(* IEC 61131-3 sources: verifaps-lib/geteta/examples/RTT_if, 5 files *)

(* ---- Preamble.st ---- *)
TYPE
    Magazin_states_t : (Green_Lamp , Init , Interstep , Magazin_Init , Magazin_Init_2 , Slider_Move_Back , Start_Magazin , Step0 , Step1 , convey);
    Stamp_states_t : (Green_Lamp , Init , Interstep , Interstep_2 , StampProcess , StampSliderBack , StampSliderForward , Stamp_Init_1 , Stamp_Init_2 , Stamp_Init_3 , Stamp_Init_4 , Start_Stamp , Step0 , Step1 , Step2);
    Crane_states_t : (Crane_Go_Up , Crane_Init , Crane_Init_2 , Crane_Lift_At_Stamp , Crane_Lift_Conveyor , Crane_Lift_Conveyor_Black , Crane_Lift_Magazin , Crane_Lift_Magazin_Metallic , Crane_Lift_NOT_Metallic_Black , Crane_Lower , Crane_On_Conveyor , Crane_On_Conveyor_Metallic , Crane_On_Conveyor_Not_Metallica_Black , Crane_On_Stamp_Metallic , Crane_On_Stamp_Stop_Black , Crane_Turn_Left_Back_To_Stamp , Crane_Turn_Left_From_Stamp , Crane_Turn_Left_Metallic , Crane_Turn_Left_NOT_Metallic , Crane_Turn_Left_NOT_Metallic_Black , Init , Interstep , Interstep_2 , Last_Workpiece_At_Stamp , Lower_Crane , Magazin_Stop , Magazin_Stop_Black , No_Workpiece_ready , Reset_interconnect , Start_Crane , Step0 , Suck_At_Stamp , TimeDelay , Turn_Right , Turn_Right_Black , pause , release , release_Black , release_Workpiece);
END_TYPE

(* ---- Code_13.st ---- *)
FUNCTION_BLOCK Main

VAR_OUTPUT  Actuator_AnalogCranePressure : INT; END_VAR
VAR_OUTPUT  Actuator_CraneLower : BOOL; END_VAR
VAR_OUTPUT  Actuator_CraneTurnClockwise : BOOL; END_VAR
VAR_OUTPUT  Actuator_CraneTurnCounterclockwise : BOOL; END_VAR
VAR_OUTPUT  Actuator_MagazinGreenLamp : BOOL; END_VAR
VAR_OUTPUT  Actuator_MagazinSlider : BOOL; END_VAR
VAR_OUTPUT  Actuator_MagazinVacuumOff : BOOL; END_VAR
VAR_OUTPUT  Actuator_MagazinVacuumOn : BOOL; END_VAR
VAR_OUTPUT  Actuator_MagazinWhiteLamp : BOOL; END_VAR
VAR_OUTPUT  Actuator_PusherY1 : BOOL; END_VAR
VAR_OUTPUT  Actuator_PusherY2 : BOOL; END_VAR
VAR_OUTPUT  Actuator_SorterConveyorTowardsCrane : BOOL; END_VAR
VAR_OUTPUT  Actuator_SorterConveyorTowardsStacker : BOOL; END_VAR
VAR_OUTPUT  Actuator_SorterGreenLampConveyor : BOOL; END_VAR
VAR_OUTPUT  Actuator_SorterWhiteLampConveyor : BOOL; END_VAR
VAR_OUTPUT  Actuator_StampGreenLamp : BOOL; END_VAR
VAR_OUTPUT  Actuator_StampPusher : BOOL; END_VAR
VAR_OUTPUT  Actuator_StampSliderMovedIn : BOOL; END_VAR
VAR_OUTPUT  Actuator_StampSliderMovedOut : BOOL; END_VAR
VAR_OUTPUT  Actuator_StampWhiteLamp : BOOL; END_VAR
VAR  Conveyor$Duration_Conveyor_Runtime : UINT := UINT#1125; END_VAR
VAR  Conveyor$Duration_Conveyor_Test : UINT := UINT#250; END_VAR
VAR  Conveyor$SFCInit : BOOL; END_VAR
VAR  Conveyor$SFCReset : BOOL; END_VAR
VAR  Conveyor$SorterConveyorTowardsCrane : BOOL; END_VAR
VAR  Conveyor$SorterConveyorTowardsStacker : BOOL; END_VAR
VAR  Conveyor$SorterGreenLampConveyor : BOOL; END_VAR
VAR  Conveyor$SorterLightbarrierCraneInterface : BOOL; END_VAR
VAR  Conveyor$SorterStartButton : BOOL; END_VAR
VAR  Conveyor$SorterSwitchManuellAutomatic : BOOL; END_VAR
VAR  Conveyor$SorterWhiteLampConveyor : BOOL; END_VAR
VAR  Conveyor$StartCommandConveyor : BOOL; END_VAR
VAR  Conveyor$StartVar : BOOL; END_VAR
VAR  Conveyor$Timer_Conveyor_Runtime$ET : USINT; END_VAR
VAR  Conveyor$Timer_Conveyor_Runtime$IN : BOOL; END_VAR
VAR  Conveyor$Timer_Conveyor_Runtime$PT : USINT; END_VAR
VAR  Conveyor$Timer_Conveyor_Runtime$Q : BOOL; END_VAR
VAR  Conveyor$Timer_Conveyor_Test$ET : USINT; END_VAR
VAR  Conveyor$Timer_Conveyor_Test$IN : BOOL; END_VAR
VAR  Conveyor$Timer_Conveyor_Test$PT : USINT; END_VAR
VAR  Conveyor$Timer_Conveyor_Test$Q : BOOL; END_VAR
VAR  Conveyor$_state : Conveyor_states_t; END_VAR
VAR  Conveyor$_transit : BOOL; END_VAR
VAR  Conveyor$interconnectConveyorStartCommand : BOOL; END_VAR
VAR  Conveyor$interconnectConveyorTerminationCommand : BOOL; END_VAR
VAR  Conveyor$interconnect_Conveyor_Runtime : BOOL; END_VAR
VAR  Conveyor$interconnect_Conveyor_Test : BOOL; END_VAR
VAR  Crane$AnalogCranePosition : INT; END_VAR
VAR  Crane$AnalogCranePressure : INT; END_VAR
VAR  Crane$CraneDown : BOOL; END_VAR
VAR  Crane$CraneLower : BOOL; END_VAR
VAR  Crane$CraneSucked : BOOL; END_VAR
VAR  Crane$CraneTurnClockwise : BOOL; END_VAR
VAR  Crane$CraneTurnCounterclockwise : BOOL; END_VAR
VAR  Crane$CraneUp : BOOL; END_VAR
VAR  Crane$Duration1 : UINT := UINT#375; END_VAR
VAR  Crane$MagazinCapacitiveSensor : BOOL; END_VAR
VAR  Crane$MagazinOpticalSensor : BOOL; END_VAR
VAR  Crane$MagazinSlider : BOOL; END_VAR
VAR  Crane$MagazinVacuumOff : BOOL; END_VAR
VAR  Crane$MagazinVacuumOn : BOOL; END_VAR
VAR  Crane$SFCInit : BOOL; END_VAR
VAR  Crane$SFCReset : BOOL; END_VAR
VAR  Crane$SliderMovedOut : BOOL; END_VAR
VAR  Crane$SliderNotMovedOut : BOOL; END_VAR
VAR  Crane$StampLowered : BOOL; END_VAR
VAR  Crane$StampSliderFilled : BOOL; END_VAR
VAR  Crane$StampSliderSensorMovedOut : BOOL; END_VAR
VAR  Crane$StartButtonMagazin : BOOL; END_VAR
VAR  Crane$StartCommandCrane : BOOL; END_VAR
VAR  Crane$StartVar : BOOL; END_VAR
VAR  Crane$TimeDelay_Timer$ET : USINT; END_VAR
VAR  Crane$TimeDelay_Timer$IN : BOOL; END_VAR
VAR  Crane$TimeDelay_Timer$PT : USINT; END_VAR
VAR  Crane$TimeDelay_Timer$Q : BOOL; END_VAR
VAR  Crane$TimeDelay_Timer_Duration : UINT := UINT#12; END_VAR
VAR  Crane$TimeDelay_Timer_interconnect : BOOL; END_VAR
VAR  Crane$Timer1$ET : USINT; END_VAR
VAR  Crane$Timer1$IN : BOOL; END_VAR
VAR  Crane$Timer1$PT : USINT; END_VAR
VAR  Crane$Timer1$Q : BOOL; END_VAR
VAR  Crane$WorkpieceReady : BOOL; END_VAR
VAR  Crane$_state : Crane_states_t; END_VAR
VAR  Crane$_transit : BOOL; END_VAR
VAR  Crane$actualtime1 : INT; END_VAR
VAR  Crane$interconnect : BOOL; END_VAR
VAR  Crane$interconnectCraneStartCommand : BOOL; END_VAR
VAR  Mag$AnalogCranePosition : INT; END_VAR
VAR  Mag$CraneDown : BOOL; END_VAR
VAR  Mag$CraneLower : BOOL; END_VAR
VAR  Mag$CraneOnConveyor : BOOL; END_VAR
VAR  Mag$CraneOnMagazin : BOOL; END_VAR
VAR  Mag$CraneSucked : BOOL; END_VAR
VAR  Mag$CraneTurnClockwise : BOOL; END_VAR
VAR  Mag$CraneTurnCounterclockwise : BOOL; END_VAR
VAR  Mag$CraneUp : BOOL; END_VAR
VAR  Mag$MagazinGreenLamp : BOOL; END_VAR
VAR  Mag$MagazinSlider : BOOL; END_VAR
VAR  Mag$MagazinVacuumOff : BOOL; END_VAR
VAR  Mag$MagazinVacuumOn : BOOL; END_VAR
VAR  Mag$MagazinWhiteLamp : BOOL; END_VAR
VAR  Mag$SFCInit : BOOL; END_VAR
VAR  Mag$SFCReset : BOOL; END_VAR
VAR  Mag$SliderMovedOut : BOOL; END_VAR
VAR  Mag$SliderNotMovedOut : BOOL; END_VAR
VAR  Mag$StartButtonMagazin : BOOL; END_VAR
VAR  Mag$StartCommandMagazin : BOOL; END_VAR
VAR  Mag$StartVar : BOOL; END_VAR
VAR  Mag$WorkpieceReady : BOOL; END_VAR
VAR  Mag$_state : Magazin_states_t; END_VAR
VAR  Mag$_transit : BOOL; END_VAR
VAR  Mag$interconnectMagazinStartCommand : BOOL; END_VAR
VAR  Pusher$Duration2 : UINT := UINT#500; END_VAR
VAR  Pusher$Duration3 : UINT := UINT#50; END_VAR
VAR  Pusher$Duration_Slide1_Black : UINT := UINT#237; END_VAR
VAR  Pusher$Duration_Slide1_Metal : UINT := UINT#75; END_VAR
VAR  Pusher$Duration_Slide1_White : UINT := UINT#75; END_VAR
VAR  Pusher$Duration_Slide2_Black : UINT := UINT#500; END_VAR
VAR  Pusher$Duration_Slide2_Metal : UINT := UINT#92; END_VAR
VAR  Pusher$Duration_Slide2_White : UINT := UINT#92; END_VAR
VAR  Pusher$Priority_Var_Black : INT := INT#3; END_VAR
VAR  Pusher$Priority_Var_Metal : INT := INT#3; END_VAR
VAR  Pusher$Priority_Var_White : INT := INT#3; END_VAR
VAR  Pusher$PusherY1 : BOOL; END_VAR
VAR  Pusher$PusherY2 : BOOL; END_VAR
VAR  Pusher$SFCInit : BOOL; END_VAR
VAR  Pusher$SFCReset : BOOL; END_VAR
VAR  Pusher$Slide1_black : INT := INT#1; END_VAR
VAR  Pusher$Slide1_metal : INT := INT#1; END_VAR
VAR  Pusher$Slide1_white : INT := INT#1; END_VAR
VAR  Pusher$Slide2_black : INT := INT#1; END_VAR
VAR  Pusher$Slide2_metal : INT := INT#1; END_VAR
VAR  Pusher$Slide2_white : INT := INT#1; END_VAR
VAR  Pusher$Slide3_black : INT := INT#1; END_VAR
VAR  Pusher$Slide3_metal : INT := INT#1; END_VAR
VAR  Pusher$Slide3_white : INT := INT#1; END_VAR
VAR  Pusher$SorterCapacitiveSensorPusher1 : BOOL; END_VAR
VAR  Pusher$SorterCapacitiveSensorPusher2 : BOOL; END_VAR
VAR  Pusher$SorterLightbarrierCraneInterface : BOOL; END_VAR
VAR  Pusher$SorterLightnessSensorPusher1 : BOOL; END_VAR
VAR  Pusher$SorterLightnessSensorPusher2 : BOOL; END_VAR
VAR  Pusher$SorterLightnessSensorPusher3 : BOOL; END_VAR
VAR  Pusher$SorterLightnesssensorCraneInterfaceInverse : BOOL; END_VAR
VAR  Pusher$SorterPusher1MovedIn : BOOL; END_VAR
VAR  Pusher$SorterPusher1MovedOut : BOOL; END_VAR
VAR  Pusher$SorterPusher2MovedIn : BOOL; END_VAR
VAR  Pusher$SorterPusher2MovedOut : BOOL; END_VAR
VAR  Pusher$SorterStartButton : BOOL; END_VAR
VAR  Pusher$StartVar : BOOL; END_VAR
VAR  Pusher$Timer2$ET : USINT; END_VAR
VAR  Pusher$Timer2$IN : BOOL; END_VAR
VAR  Pusher$Timer2$PT : USINT; END_VAR
VAR  Pusher$Timer2$Q : BOOL; END_VAR
VAR  Pusher$Timer3$ET : USINT; END_VAR
VAR  Pusher$Timer3$IN : BOOL; END_VAR
VAR  Pusher$Timer3$PT : USINT; END_VAR
VAR  Pusher$Timer3$Q : BOOL; END_VAR
VAR  Pusher$Timer_Slide1_Black$ET : USINT; END_VAR
VAR  Pusher$Timer_Slide1_Black$IN : BOOL; END_VAR
VAR  Pusher$Timer_Slide1_Black$PT : USINT; END_VAR
VAR  Pusher$Timer_Slide1_Black$Q : BOOL; END_VAR
VAR  Pusher$Timer_Slide1_Metal$ET : USINT; END_VAR
VAR  Pusher$Timer_Slide1_Metal$IN : BOOL; END_VAR
VAR  Pusher$Timer_Slide1_Metal$PT : USINT; END_VAR
VAR  Pusher$Timer_Slide1_Metal$Q : BOOL; END_VAR
VAR  Pusher$Timer_Slide1_White$ET : USINT; END_VAR
VAR  Pusher$Timer_Slide1_White$IN : BOOL; END_VAR
VAR  Pusher$Timer_Slide1_White$PT : USINT; END_VAR
VAR  Pusher$Timer_Slide1_White$Q : BOOL; END_VAR
VAR  Pusher$Timer_Slide2_Black$ET : USINT; END_VAR
VAR  Pusher$Timer_Slide2_Black$IN : BOOL; END_VAR
VAR  Pusher$Timer_Slide2_Black$PT : USINT; END_VAR
VAR  Pusher$Timer_Slide2_Black$Q : BOOL; END_VAR
VAR  Pusher$Timer_Slide2_Metal$ET : USINT; END_VAR
VAR  Pusher$Timer_Slide2_Metal$IN : BOOL; END_VAR
VAR  Pusher$Timer_Slide2_Metal$PT : USINT; END_VAR
VAR  Pusher$Timer_Slide2_Metal$Q : BOOL; END_VAR
VAR  Pusher$Timer_Slide2_White$ET : USINT; END_VAR
VAR  Pusher$Timer_Slide2_White$IN : BOOL; END_VAR
VAR  Pusher$Timer_Slide2_White$PT : USINT; END_VAR
VAR  Pusher$Timer_Slide2_White$Q : BOOL; END_VAR
VAR  Pusher$_state : Pusher_states_t; END_VAR
VAR  Pusher$_transit : BOOL; END_VAR
VAR  Pusher$interconnect2 : BOOL; END_VAR
VAR  Pusher$interconnect3 : BOOL; END_VAR
VAR  Pusher$interconnect_Slide1_Black : BOOL; END_VAR
VAR  Pusher$interconnect_Slide1_Metal : BOOL; END_VAR
VAR  Pusher$interconnect_Slide1_White : BOOL; END_VAR
VAR  Pusher$interconnect_Slide2_Black : BOOL; END_VAR
VAR  Pusher$interconnect_Slide2_Metal : BOOL; END_VAR
VAR  Pusher$interconnect_Slide2_White : BOOL; END_VAR
VAR_INPUT  Sensor_AnalogCranePosition : INT; END_VAR
VAR_INPUT  Sensor_CraneDown : BOOL; END_VAR
VAR_INPUT  Sensor_CraneOnConveyor : BOOL; END_VAR
VAR_INPUT  Sensor_CraneOnMagazin : BOOL; END_VAR
VAR_INPUT  Sensor_CranePosition : BOOL; END_VAR
VAR_INPUT  Sensor_CranePositionStamp : BOOL; END_VAR
VAR_INPUT  Sensor_CraneSucked : BOOL; END_VAR
VAR_INPUT  Sensor_CraneUp : BOOL; END_VAR
VAR_INPUT  Sensor_MagazinCapacitiveSensor : BOOL; END_VAR
VAR_INPUT  Sensor_MagazinEmergencyStop : BOOL; END_VAR
VAR_INPUT  Sensor_MagazinOpticalSensor : BOOL; END_VAR
VAR_INPUT  Sensor_MagazinSwitchManuellAutomatic : BOOL; END_VAR
VAR_INPUT  Sensor_SliderMovedOut : BOOL; END_VAR
VAR_INPUT  Sensor_SliderNotMovedOut : BOOL; END_VAR
VAR_INPUT  Sensor_SorterCapacitiveSensorPusher1 : BOOL; END_VAR
VAR_INPUT  Sensor_SorterCapacitiveSensorPusher2 : BOOL; END_VAR
VAR_INPUT  Sensor_SorterEmergencyStop : BOOL; END_VAR
VAR_INPUT  Sensor_SorterLightbarrierCraneInterface : BOOL; END_VAR
VAR_INPUT  Sensor_SorterLightnessSensorPusher1 : BOOL; END_VAR
VAR_INPUT  Sensor_SorterLightnessSensorPusher2 : BOOL; END_VAR
VAR_INPUT  Sensor_SorterLightnessSensorPusher3 : BOOL; END_VAR
VAR_INPUT  Sensor_SorterLightnesssensorCraneInterfaceInverse : BOOL; END_VAR
VAR_INPUT  Sensor_SorterPusher1MovedIn : BOOL; END_VAR
VAR_INPUT  Sensor_SorterPusher1MovedOut : BOOL; END_VAR
VAR_INPUT  Sensor_SorterPusher2MovedIn : BOOL; END_VAR
VAR_INPUT  Sensor_SorterPusher2MovedOut : BOOL; END_VAR
VAR_INPUT  Sensor_SorterStartButton : BOOL; END_VAR
VAR_INPUT  Sensor_SorterSwitchManuellAutomatic : BOOL; END_VAR
VAR_INPUT  Sensor_StampEmergencyStop : BOOL; END_VAR
VAR_INPUT  Sensor_StampLowered : BOOL; END_VAR
VAR_INPUT  Sensor_StampSliderFilled : BOOL; END_VAR
VAR_INPUT  Sensor_StampSliderSensorMovedIn : BOOL; END_VAR
VAR_INPUT  Sensor_StampSliderSensorMovedOut : BOOL; END_VAR
VAR_INPUT  Sensor_StampStartButton : BOOL; END_VAR
VAR_INPUT  Sensor_StampSwitchManuellAutomatic : BOOL; END_VAR
VAR_INPUT  Sensor_StampUp : BOOL; END_VAR
VAR_INPUT  Sensor_StartButtonMagazin : BOOL; END_VAR
VAR_INPUT  Sensor_WorkpieceReady : BOOL; END_VAR
VAR  Stamp$AnalogCranePosition : INT; END_VAR
VAR  Stamp$CraneDown : BOOL; END_VAR
VAR  Stamp$CraneOnConveyor : BOOL; END_VAR
VAR  Stamp$CranePositionStamp : BOOL; END_VAR
VAR  Stamp$CraneSucked : BOOL; END_VAR
VAR  Stamp$CraneUp : BOOL; END_VAR
        VAR  Stamp$Duration : UINT := UINT#125; END_VAR

VAR  Stamp$SFCInit : BOOL; END_VAR
VAR  Stamp$SFCReset : BOOL; END_VAR
VAR  Stamp$StampGreenLamp : BOOL; END_VAR
VAR  Stamp$StampLowered : BOOL; END_VAR
VAR  Stamp$StampPressure : BOOL; END_VAR
VAR  Stamp$StampPusher : BOOL; END_VAR
VAR  Stamp$StampSliderFilled : BOOL; END_VAR
VAR  Stamp$StampSliderMovedIn : BOOL; END_VAR
VAR  Stamp$StampSliderMovedOut : BOOL; END_VAR
VAR  Stamp$StampSliderSensorMovedIn : BOOL; END_VAR
VAR  Stamp$StampSliderSensorMovedOut : BOOL; END_VAR
VAR  Stamp$StampStartButton : BOOL; END_VAR
VAR  Stamp$StampUp : BOOL; END_VAR
VAR  Stamp$StampWhiteLamp : BOOL; END_VAR
VAR  Stamp$StartCommandStamp : BOOL; END_VAR
VAR  Stamp$StartVar : BOOL; END_VAR
VAR  Stamp$Timer$ET : USINT; END_VAR
VAR  Stamp$Timer$IN : BOOL; END_VAR
VAR  Stamp$Timer$PT : USINT; END_VAR
VAR  Stamp$Timer$Q : BOOL; END_VAR
VAR  Stamp$_state : Stamp_states_t; END_VAR
VAR  Stamp$_transit : BOOL; END_VAR
VAR  Stamp$interconnect : BOOL; END_VAR
VAR  Stamp$interconnectStampStartCommand : BOOL; END_VAR

VAR  DIAGNOSIS_ACTIVE : BOOL; END_VAR

VAR_INPUT PARAMETER_CRANE_PRESSURE_METALLIC : INT := INT#6000; END_VAR
VAR_INPUT PARAMETER_CRANE_PRESSURE_WHITE : INT := INT#7000; END_VAR

// impl
Mag$SliderNotMovedOut := Sensor_SliderNotMovedOut;
Mag$SliderMovedOut := Sensor_SliderMovedOut;
Mag$CraneOnMagazin := Sensor_CraneOnMagazin;
Mag$CraneDown := Sensor_CraneDown;
Mag$CraneUp := Sensor_CraneUp;
Mag$CraneOnConveyor := Sensor_CraneOnConveyor;
Mag$WorkpieceReady := Sensor_WorkpieceReady;
Mag$AnalogCranePosition := Sensor_AnalogCranePosition;
Mag$StartButtonMagazin := Sensor_StartButtonMagazin;
Actuator_MagazinSlider := Mag$MagazinSlider;
Actuator_MagazinGreenLamp := Mag$MagazinGreenLamp;
Crane$CraneUp := Sensor_CraneUp;
Crane$CraneDown := Sensor_CraneDown;
Crane$CraneSucked := Sensor_CraneSucked;
Crane$MagazinCapacitiveSensor := Sensor_MagazinCapacitiveSensor;
Crane$SliderMovedOut := Sensor_SliderMovedOut;
Crane$WorkpieceReady := Sensor_WorkpieceReady;
Crane$MagazinOpticalSensor := Sensor_MagazinOpticalSensor;
Crane$StampSliderFilled := Sensor_StampSliderFilled;
Crane$StampSliderSensorMovedOut := Sensor_StampSliderSensorMovedOut;
Crane$StampLowered := Sensor_StampLowered;
Crane$AnalogCranePosition := Sensor_AnalogCranePosition;
Crane$StartButtonMagazin := Sensor_StartButtonMagazin;

//Diagnosis
// old: Actuator_AnalogCranePressure
// new: Crane$AnalogCranePressure;
Actuator_CraneTurnCounterclockwise := Crane$CraneTurnCounterclockwise;
Actuator_CraneTurnClockwise := Crane$CraneTurnClockwise;

IF DIAGNOSIS_ACTIVE THEN
        IF Sensor_CraneSucked AND (Crane$AnalogCranePressure <= 0 OR Crane$AnalogCranePressure > 10000) THEN
                Actuator_CraneTurnCounterclockwise := FALSE;
                Actuator_CraneTurnClockwise := FALSE;
        END_IF
END_IF

//End of Diagnosis

Actuator_CraneLower := Crane$CraneLower;
Actuator_MagazinVacuumOff := Crane$MagazinVacuumOff;
Actuator_MagazinVacuumOn := Crane$MagazinVacuumOn;
Actuator_AnalogCranePressure := Crane$AnalogCranePressure;
Stamp$StampSliderSensorMovedOut := Sensor_StampSliderSensorMovedOut;
Stamp$StampSliderSensorMovedIn := Sensor_StampSliderSensorMovedIn;
Stamp$StampSliderFilled := Sensor_StampSliderFilled;
Stamp$StampUp := Sensor_StampUp;
Stamp$StampLowered := Sensor_StampLowered;
Stamp$CraneDown := Sensor_CraneDown;
Stamp$CraneUp := Sensor_CraneUp;
Stamp$CraneSucked := Sensor_CraneSucked;
Stamp$CranePositionStamp := Sensor_CranePositionStamp;
Stamp$CraneOnConveyor := Sensor_CraneOnConveyor;
Stamp$AnalogCranePosition := Sensor_AnalogCranePosition;
Stamp$StampStartButton := Sensor_StampStartButton;
Actuator_StampSliderMovedOut := Stamp$StampSliderMovedOut;
Actuator_StampSliderMovedIn := Stamp$StampSliderMovedIn;
Actuator_StampWhiteLamp := Stamp$StampWhiteLamp;
Actuator_StampPusher := Stamp$StampPusher;
Actuator_StampGreenLamp := Stamp$StampGreenLamp;
Conveyor$SorterStartButton := Sensor_SorterStartButton;
Conveyor$SorterSwitchManuellAutomatic := Sensor_SorterSwitchManuellAutomatic;
Conveyor$SorterLightbarrierCraneInterface := Sensor_SorterLightbarrierCraneInterface;
Actuator_SorterConveyorTowardsStacker := Conveyor$SorterConveyorTowardsStacker;
Actuator_SorterConveyorTowardsCrane := Conveyor$SorterConveyorTowardsCrane;
Actuator_SorterGreenLampConveyor := Conveyor$SorterGreenLampConveyor;
Actuator_SorterWhiteLampConveyor := Conveyor$SorterWhiteLampConveyor;
Pusher$SorterLightnesssensorCraneInterfaceInverse := Sensor_SorterLightnesssensorCraneInterfaceInverse;
Pusher$SorterLightbarrierCraneInterface := Sensor_SorterLightbarrierCraneInterface;
Pusher$SorterCapacitiveSensorPusher1 := Sensor_SorterCapacitiveSensorPusher1;
Pusher$SorterLightnessSensorPusher1 := Sensor_SorterLightnessSensorPusher1;
Pusher$SorterCapacitiveSensorPusher2 := Sensor_SorterCapacitiveSensorPusher2;
Pusher$SorterLightnessSensorPusher2 := Sensor_SorterLightnessSensorPusher2;
Pusher$SorterLightnessSensorPusher3 := Sensor_SorterLightnessSensorPusher3;
Pusher$SorterPusher1MovedOut := Sensor_SorterPusher1MovedOut;
Pusher$SorterPusher1MovedIn := Sensor_SorterPusher1MovedIn;
Pusher$SorterPusher2MovedOut := Sensor_SorterPusher2MovedOut;
Pusher$SorterPusher2MovedIn := Sensor_SorterPusher2MovedIn;
Pusher$SorterStartButton := Sensor_SorterStartButton;
Actuator_PusherY1 := Pusher$PusherY1;
Actuator_PusherY2 := Pusher$PusherY2;

IF ((Sensor_SorterEmergencyStop AND Sensor_StampEmergencyStop) AND Sensor_MagazinEmergencyStop) THEN
    CASE Mag$_state OF
        Magazin_states_t#Green_Lamp:
            Mag$_transit := FALSE;
            Mag$MagazinGreenLamp := TRUE;
            Mag$interconnectMagazinStartCommand := FALSE;
            IF TRUE THEN
                Mag$_transit := TRUE;
                Mag$_state := Magazin_states_t#Magazin_Init;
            END_IF

        Magazin_states_t#Init:
            Mag$_transit := FALSE;
            IF TRUE THEN
                Mag$_transit := TRUE;
                Mag$_state := Magazin_states_t#Start_Magazin;
            END_IF

        Magazin_states_t#Interstep:
            Mag$_transit := FALSE;
            Mag$StartCommandMagazin := TRUE;
            IF Mag$StartVar THEN
                Mag$_transit := TRUE;
                Mag$_state := Magazin_states_t#convey;
            END_IF

        Magazin_states_t#Magazin_Init:
            Mag$_transit := FALSE;
            Mag$MagazinSlider := TRUE;
            IF TRUE THEN
                Mag$_transit := TRUE;
                Mag$_state := Magazin_states_t#Magazin_Init_2;
            END_IF

        Magazin_states_t#Magazin_Init_2:
            Mag$_transit := FALSE;
            Mag$MagazinSlider := FALSE;
            IF TRUE THEN
                Mag$_transit := TRUE;
                Mag$_state := Magazin_states_t#Interstep;
            END_IF

        Magazin_states_t#Slider_Move_Back:
            Mag$_transit := FALSE;
            IF ((Mag$SliderMovedOut = TRUE) AND (Mag$SliderNotMovedOut = FALSE)) THEN
                Mag$MagazinSlider := FALSE;
            END_IF
            IF Mag$CraneUp THEN
                Mag$_transit := TRUE;
                Mag$_state := Magazin_states_t#Step1;
            END_IF

        Magazin_states_t#Start_Magazin:
            Mag$_transit := FALSE;
            Mag$MagazinSlider := FALSE;
            Mag$MagazinGreenLamp := FALSE;
            Mag$StartVar := FALSE;
            Mag$StartCommandMagazin := FALSE;
            IF (Mag$StartButtonMagazin = TRUE) THEN
                Mag$interconnectMagazinStartCommand := TRUE;
            END_IF
            IF Mag$interconnectMagazinStartCommand THEN
                Mag$_transit := TRUE;
                Mag$_state := Magazin_states_t#Green_Lamp;
            END_IF

        Magazin_states_t#Step0:
            Mag$_transit := FALSE;
            IF Mag$CraneDown THEN
                Mag$_transit := TRUE;
                Mag$_state := Magazin_states_t#Slider_Move_Back;
            END_IF

        Magazin_states_t#Step1:
            Mag$_transit := FALSE;
            IF ((Mag$AnalogCranePosition > INT#16160) AND (Mag$AnalogCranePosition < INT#16260)) THEN
                Mag$_transit := TRUE;
                Mag$_state := Magazin_states_t#Interstep;
            END_IF

        Magazin_states_t#convey:
            Mag$_transit := FALSE;
            IF Mag$SliderNotMovedOut THEN
                Mag$MagazinSlider := TRUE;
            END_IF
            IF ((Mag$AnalogCranePosition > INT#24290) AND (Mag$AnalogCranePosition < INT#24390)) THEN
                Mag$_transit := TRUE;
                Mag$_state := Magazin_states_t#Step0;
            END_IF

            END_CASE
    CASE Crane$_state OF
        Crane_states_t#Crane_Go_Up:
            Crane$_transit := FALSE;
            Crane$CraneLower := FALSE;
            IF Crane$CraneUp THEN
                Crane$_transit := TRUE;
                Crane$_state := Crane_states_t#Step3;
            END_IF

        Crane_states_t#Crane_Go_Up_White:
            Crane$_transit := FALSE;
            Crane$CraneLower := FALSE;
            IF Crane$CraneUp THEN
                Crane$_transit := TRUE;
                Crane$_state := Crane_states_t#Step3;
            END_IF

        Crane_states_t#Crane_Init:
            Crane$_transit := FALSE;
            Crane$CraneLower := TRUE;
            Crane$interconnectCraneStartCommand := FALSE;
            Crane$AnalogCranePressure := PARAMETER_CRANE_PRESSURE_METALLIC;
            IF Crane$CraneDown THEN
                Crane$_transit := TRUE;
                Crane$_state := Crane_states_t#Crane_Init_2;
            END_IF

        Crane_states_t#Crane_Init_2:
            Crane$_transit := FALSE;
            Crane$CraneLower := FALSE;
            IF Crane$CraneUp THEN
                Crane$_transit := TRUE;
                Crane$_state := Crane_states_t#Interstep;
            END_IF

        Crane_states_t#Crane_Lift_At_Stamp:
            Crane$_transit := FALSE;
            Crane$CraneLower := FALSE;
            IF Crane$CraneUp THEN
                Crane$_transit := TRUE;
                Crane$_state := Crane_states_t#Crane_Turn_Left_From_Stamp;
            END_IF

        Crane_states_t#Crane_Lift_At_Stamp2:
            Crane$_transit := FALSE;
            Crane$CraneLower := FALSE;
            Crane$AnalogCranePressure := INT#0;
            IF Crane$CraneUp THEN
                Crane$_transit := TRUE;
                Crane$_state := Crane_states_t#Crane_Turn_Right_From_Stamp;
            END_IF

        Crane_states_t#Crane_Lift_Conveyor:
            Crane$_transit := FALSE;
            Crane$CraneLower := FALSE;
            IF TRUE THEN
                Crane$_transit := TRUE;
                Crane$_state := Crane_states_t#Interstep;
            END_IF

        Crane_states_t#Crane_Lift_Conveyor2:
            Crane$_transit := FALSE;
            Crane$CraneLower := FALSE;
            IF TRUE THEN
                Crane$_transit := TRUE;
                Crane$_state := Crane_states_t#Interstep;
            END_IF

        Crane_states_t#Crane_Lift_Conveyor_Black:
            Crane$_transit := FALSE;
            Crane$CraneLower := FALSE;
            IF Crane$CraneUp THEN
                Crane$_transit := TRUE;
                Crane$_state := Crane_states_t#Crane_Turn_Left_Back_To_Stamp;
            END_IF

        Crane_states_t#Crane_Lift_Magazin:
            Crane$_transit := FALSE;
            Crane$CraneLower := FALSE;
            IF Crane$CraneUp THEN
                Crane$_transit := TRUE;
                Crane$_state := Crane_states_t#Crane_Turn_Left_NOT_Metallic;
            END_IF

        Crane_states_t#Crane_Lift_Magazin_Metallic:
            Crane$_transit := FALSE;
            Crane$CraneLower := FALSE;
            IF Crane$CraneUp THEN
                Crane$_transit := TRUE;
                Crane$_state := Crane_states_t#Crane_Turn_Left_Metallic;
            END_IF

        Crane_states_t#Crane_Lift_Magazin_White:
            Crane$_transit := FALSE;
            Crane$CraneLower := FALSE;
            IF Crane$CraneUp THEN
                Crane$_transit := TRUE;
                Crane$_state := Crane_states_t#Crane_Turn_Left_White;
            END_IF

        Crane_states_t#Crane_Lift_NOT_Metallic_Black:
            Crane$_transit := FALSE;
            Crane$CraneLower := FALSE;
            IF Crane$CraneUp THEN
                Crane$_transit := TRUE;
                Crane$_state := Crane_states_t#Crane_Turn_Left_NOT_Metallic_Black;
            END_IF

        Crane_states_t#Crane_Lower:
            Crane$_transit := FALSE;
            Crane$MagazinVacuumOn := TRUE;
            Crane$MagazinVacuumOff := FALSE;
            Crane$CraneLower := TRUE;
            Crane$AnalogCranePressure := INT#0;
            IF Crane$CraneSucked THEN
                Crane$_transit := TRUE;
                Crane$_state := Crane_states_t#Step0;
            END_IF

        Crane_states_t#Crane_On_Conveyor:
            Crane$_transit := FALSE;
            Crane$CraneTurnCounterclockwise := FALSE;
            Crane$CraneTurnClockwise := FALSE;
            Crane$CraneLower := TRUE;
            IF Crane$CraneDown THEN
                Crane$_transit := TRUE;
                Crane$_state := Crane_states_t#release;
            END_IF

        Crane_states_t#Crane_On_Conveyor_Metallic:
            Crane$_transit := FALSE;
            Crane$CraneTurnCounterclockwise := FALSE;
            Crane$CraneTurnClockwise := FALSE;
            Crane$CraneLower := TRUE;
            IF Crane$CraneDown THEN
                Crane$_transit := TRUE;
                Crane$_state := Crane_states_t#release;
            END_IF

        Crane_states_t#Crane_On_Conveyor_Metallic2:
            Crane$_transit := FALSE;
            Crane$CraneTurnCounterclockwise := FALSE;
            Crane$CraneTurnClockwise := FALSE;
            Crane$CraneLower := TRUE;
            IF Crane$CraneDown THEN
                Crane$_transit := TRUE;
                Crane$_state := Crane_states_t#release2;
            END_IF

        Crane_states_t#Crane_On_Conveyor_Not_Metallica_Black:
            Crane$_transit := FALSE;
            Crane$CraneTurnCounterclockwise := FALSE;
            Crane$CraneTurnClockwise := FALSE;
            Crane$CraneLower := TRUE;
            IF Crane$CraneDown THEN
                Crane$_transit := TRUE;
                Crane$_state := Crane_states_t#release_Black;
            END_IF

        Crane_states_t#Crane_On_Stamp_Metallic:
            Crane$_transit := FALSE;
            Crane$CraneTurnCounterclockwise := FALSE;
            Crane$CraneTurnClockwise := FALSE;
            Crane$CraneLower := TRUE;
            IF Crane$CraneDown THEN
                Crane$_transit := TRUE;
                Crane$_state := Crane_states_t#release_Workpiece;
            END_IF

        Crane_states_t#Crane_On_Stamp_Metallic2:
            Crane$_transit := FALSE;
            Crane$CraneTurnCounterclockwise := FALSE;
            Crane$CraneTurnClockwise := FALSE;
            IF Crane$StampLowered THEN
                Crane$_transit := TRUE;
                Crane$_state := Crane_states_t#Interstep_4;
            END_IF

        Crane_states_t#Crane_On_Stamp_Metallic2_Lower:
            Crane$_transit := FALSE;
            Crane$CraneLower := TRUE;
            IF Crane$CraneDown THEN
                Crane$_transit := TRUE;
                Crane$_state := Crane_states_t#Suck_At_Stamp2;
            END_IF

        Crane_states_t#Crane_On_Stamp_Stop_Black:
            Crane$_transit := FALSE;
            Crane$CraneTurnClockwise := FALSE;
            Crane$CraneTurnCounterclockwise := FALSE;
            IF TRUE THEN
                Crane$_transit := TRUE;
                Crane$_state := Crane_states_t#Reset_interconnect;
            END_IF

        Crane_states_t#Crane_On_Stamp_White:
            Crane$_transit := FALSE;
            Crane$CraneTurnCounterclockwise := FALSE;
            Crane$CraneTurnClockwise := FALSE;
            Crane$CraneLower := TRUE;
            IF Crane$CraneDown THEN
                Crane$_transit := TRUE;
                Crane$_state := Crane_states_t#release_Workpiece_White;
            END_IF

        Crane_states_t#Crane_Turn_Left_Back_To_Stamp:
            Crane$_transit := FALSE;
            Crane$CraneTurnCounterclockwise := TRUE;
            Crane$CraneTurnClockwise := FALSE;
            IF ((Crane$AnalogCranePosition > INT#8160) AND (Crane$AnalogCranePosition < INT#8260)) THEN
                Crane$_transit := TRUE;
                Crane$_state := Crane_states_t#Crane_On_Stamp_Stop_Black;
            END_IF

        Crane_states_t#Crane_Turn_Left_From_Stamp:
            Crane$_transit := FALSE;
            Crane$CraneTurnClockwise := TRUE;
            Crane$CraneTurnCounterclockwise := FALSE;
            IF ((Crane$AnalogCranePosition > INT#16060) AND (Crane$AnalogCranePosition < INT#16160)) THEN
                Crane$_transit := TRUE;
                Crane$_state := Crane_states_t#Crane_On_Conveyor_Metallic;
            END_IF

        Crane_states_t#Crane_Turn_Left_Metallic:
            Crane$_transit := FALSE;
            Crane$CraneTurnCounterclockwise := TRUE;
            Crane$CraneTurnClockwise := FALSE;
            IF ((Crane$AnalogCranePosition > INT#8160) AND (Crane$AnalogCranePosition < INT#8260)) THEN
                Crane$_transit := TRUE;
                Crane$_state := Crane_states_t#Crane_On_Stamp_Metallic;
            END_IF

        Crane_states_t#Crane_Turn_Left_Metallic2:
            Crane$_transit := FALSE;
            Crane$CraneTurnCounterclockwise := TRUE;
            Crane$CraneTurnClockwise := FALSE;
            IF ((Crane$AnalogCranePosition > INT#8160) AND (Crane$AnalogCranePosition < INT#8260)) THEN
                Crane$_transit := TRUE;
                Crane$_state := Crane_states_t#Crane_On_Stamp_Metallic2;
            END_IF

        Crane_states_t#Crane_Turn_Left_NOT_Metallic:
            Crane$_transit := FALSE;
            Crane$CraneTurnCounterclockwise := TRUE;
            Crane$CraneTurnClockwise := FALSE;
            IF ((Crane$AnalogCranePosition > INT#16160) AND (Crane$AnalogCranePosition < INT#16260)) THEN
                Crane$_transit := TRUE;
                Crane$_state := Crane_states_t#Crane_On_Conveyor;
            END_IF

        Crane_states_t#Crane_Turn_Left_NOT_Metallic_Black:
            Crane$_transit := FALSE;
            Crane$CraneTurnCounterclockwise := TRUE;
            Crane$CraneTurnClockwise := FALSE;
            IF ((Crane$AnalogCranePosition > INT#16160) AND (Crane$AnalogCranePosition < INT#16260)) THEN
                Crane$_transit := TRUE;
                Crane$_state := Crane_states_t#Crane_On_Conveyor_Not_Metallica_Black;
            END_IF

        Crane_states_t#Crane_Turn_Left_White:
            Crane$_transit := FALSE;
            Crane$CraneTurnCounterclockwise := TRUE;
            Crane$CraneTurnClockwise := FALSE;
            IF ((Crane$AnalogCranePosition > INT#8160) AND (Crane$AnalogCranePosition < INT#8260)) THEN
                Crane$_transit := TRUE;
                Crane$_state := Crane_states_t#Crane_On_Stamp_White;
            END_IF

        Crane_states_t#Crane_Turn_Right_From_Stamp:
            Crane$_transit := FALSE;
            Crane$CraneTurnClockwise := TRUE;
            Crane$CraneTurnCounterclockwise := FALSE;
            IF ((Crane$AnalogCranePosition > INT#16160) AND (Crane$AnalogCranePosition < INT#16260)) THEN
                Crane$_transit := TRUE;
                Crane$_state := Crane_states_t#Crane_On_Conveyor_Metallic2;
            END_IF

        Crane_states_t#Init:
            Crane$_transit := FALSE;
            IF TRUE THEN
                Crane$_transit := TRUE;
                Crane$_state := Crane_states_t#Start_Crane;
            END_IF

        Crane_states_t#Interstep:
            Crane$_transit := FALSE;
            Crane$StartCommandCrane := TRUE;
            IF Crane$StartVar THEN
                Crane$_transit := TRUE;
                Crane$_state := Crane_states_t#Interstep_2;
            END_IF

        Crane_states_t#Interstep_2:
            Crane$_transit := FALSE;
            IF Crane$SliderMovedOut THEN
                Crane$_transit := TRUE;
                Crane$_state := Crane_states_t#TimeDelay;
            END_IF

        Crane_states_t#Interstep_3:
            Crane$_transit := FALSE;
            IF NOT Crane$WorkpieceReady THEN
                Crane$_transit := TRUE;
                Crane$_state := Crane_states_t#No_Workpiece_ready;
            ELSEIF Crane$WorkpieceReady THEN
                Crane$_transit := TRUE;
                Crane$_state := Crane_states_t#Turn_Right;
            END_IF

        Crane_states_t#Interstep_4:
            Crane$_transit := FALSE;
            IF Crane$StampSliderSensorMovedOut THEN
                Crane$_transit := TRUE;
                Crane$_state := Crane_states_t#Crane_On_Stamp_Metallic2_Lower;
            END_IF

        Crane_states_t#Lower_Crane:
            Crane$_transit := FALSE;
            Crane$CraneLower := TRUE;
            IF Crane$CraneDown THEN
                Crane$_transit := TRUE;
                Crane$_state := Crane_states_t#Suck_At_Stamp;
            END_IF

        Crane_states_t#Magazin_Stop:
            Crane$_transit := FALSE;
            Crane$CraneTurnClockwise := FALSE;
            Crane$CraneTurnCounterclockwise := FALSE;
            IF TRUE THEN
                Crane$_transit := TRUE;
                Crane$_state := Crane_states_t#Crane_Lower;
            END_IF

        Crane_states_t#Magazin_Stop_Black:
            Crane$_transit := FALSE;
            Crane$CraneTurnClockwise := FALSE;
            Crane$CraneTurnCounterclockwise := FALSE;
            Crane$MagazinVacuumOn := TRUE;
            Crane$MagazinVacuumOff := FALSE;
            Crane$CraneLower := TRUE;
            IF Crane$CraneSucked THEN
                Crane$_transit := TRUE;
                Crane$_state := Crane_states_t#Crane_Lift_NOT_Metallic_Black;
            END_IF

        Crane_states_t#Magazin_Stop_Final:
            Crane$_transit := FALSE;
            Crane$CraneTurnClockwise := FALSE;
            Crane$CraneTurnCounterclockwise := FALSE;
            IF TRUE THEN
                Crane$_transit := TRUE;
                Crane$_state := Crane_states_t#Start_Crane;
            END_IF

        Crane_states_t#No_Workpiece_ready:
            Crane$_transit := FALSE;
            Crane$MagazinVacuumOn := FALSE;
            Crane$MagazinVacuumOff := FALSE;
            Crane$CraneLower := FALSE;
            IF Crane$StampSliderFilled THEN
                Crane$_transit := TRUE;
                Crane$_state := Crane_states_t#Crane_Turn_Left_Metallic2;
            ELSEIF NOT Crane$StampSliderFilled THEN
                Crane$_transit := TRUE;
                Crane$_state := Crane_states_t#Turn_Right_Final;
            END_IF

        Crane_states_t#Reset_interconnect:
            Crane$_transit := FALSE;
            Crane$interconnect := FALSE;
            Crane$Timer1$IN := FALSE;
            Crane$Timer1$PT := USINT#0;
            IF Crane$Timer1$IN THEN
                Crane$Timer1$Q := (Crane$Timer1$ET = USINT#0);
                IF (Crane$Timer1$ET > USINT#0) THEN
                    Crane$Timer1$ET := (Crane$Timer1$ET - USINT#1);
                ELSE
                    Crane$Timer1$ET := USINT#0;
                END_IF
            ELSE
                Crane$Timer1$Q := FALSE;
                Crane$Timer1$ET := Crane$Timer1$PT;
            END_IF
            IF Crane$SliderMovedOut THEN
                Crane$_transit := TRUE;
                Crane$_state := Crane_states_t#Lower_Crane;
            END_IF

        Crane_states_t#Stamp_Pressure_Profile_Set_Metallic:
            Crane$_transit := FALSE;
            Crane$AnalogCranePressure := PARAMETER_CRANE_PRESSURE_METALLIC;
            IF TRUE THEN
                Crane$_transit := TRUE;
                Crane$_state := Crane_states_t#Crane_Lift_Magazin_Metallic;
            END_IF

        Crane_states_t#Stamp_Pressure_Profile_Set_White:
            Crane$_transit := FALSE;
            Crane$AnalogCranePressure := PARAMETER_CRANE_PRESSURE_WHITE;
            IF TRUE THEN
                Crane$_transit := TRUE;
                Crane$_state := Crane_states_t#Crane_Lift_Magazin_White;
            END_IF

        Crane_states_t#Start_Crane:
            Crane$_transit := FALSE;
            Crane$CraneLower := FALSE;
            Crane$MagazinVacuumOff := FALSE;
            Crane$MagazinVacuumOn := FALSE;
            Crane$CraneTurnCounterclockwise := FALSE;
            Crane$CraneTurnClockwise := FALSE;
            Crane$AnalogCranePressure := INT#0;
            Crane$StartVar := FALSE;
            Crane$StartCommandCrane := FALSE;
            IF (Crane$StartButtonMagazin = TRUE) THEN
                Crane$interconnectCraneStartCommand := TRUE;
            END_IF
            IF Crane$interconnectCraneStartCommand THEN
                Crane$_transit := TRUE;
                Crane$_state := Crane_states_t#Crane_Init;
            END_IF

        Crane_states_t#Step0:
            Crane$_transit := FALSE;
            IF (Crane$MagazinCapacitiveSensor AND Crane$MagazinOpticalSensor) THEN
                Crane$_transit := TRUE;
                Crane$_state := Crane_states_t#Stamp_Pressure_Profile_Set_Metallic;
            ELSEIF (NOT Crane$MagazinCapacitiveSensor AND Crane$MagazinOpticalSensor) THEN
                Crane$_transit := TRUE;
                Crane$_state := Crane_states_t#Stamp_Pressure_Profile_Set_White;
            ELSEIF (NOT Crane$MagazinCapacitiveSensor AND NOT Crane$MagazinOpticalSensor) THEN
                Crane$_transit := TRUE;
                Crane$_state := Crane_states_t#Crane_Lift_Magazin;
            END_IF

        Crane_states_t#Step2:
            Crane$_transit := FALSE;
            IF (Crane$MagazinCapacitiveSensor OR Crane$MagazinOpticalSensor) THEN
                Crane$_transit := TRUE;
                Crane$_state := Crane_states_t#pause;
            ELSEIF (NOT Crane$MagazinCapacitiveSensor AND NOT Crane$MagazinOpticalSensor) THEN
                Crane$_transit := TRUE;
                Crane$_state := Crane_states_t#Turn_Right_Black;
            END_IF

        Crane_states_t#Step3:
            Crane$_transit := FALSE;
            IF NOT Crane$WorkpieceReady THEN
                Crane$_transit := TRUE;
                Crane$_state := Crane_states_t#Step4;
            ELSEIF Crane$WorkpieceReady THEN
                Crane$_transit := TRUE;
                Crane$_state := Crane_states_t#Step2;
            END_IF

        Crane_states_t#Step4:
            Crane$_transit := FALSE;
            IF TRUE THEN
                Crane$_transit := TRUE;
                Crane$_state := Crane_states_t#Interstep;
            END_IF

        Crane_states_t#Suck_At_Stamp:
            Crane$_transit := FALSE;
            Crane$MagazinVacuumOn := TRUE;
            Crane$MagazinVacuumOff := FALSE;
            IF Crane$CraneSucked THEN
                Crane$_transit := TRUE;
                Crane$_state := Crane_states_t#Crane_Lift_At_Stamp;
            END_IF

        Crane_states_t#Suck_At_Stamp2:
            Crane$_transit := FALSE;
            Crane$MagazinVacuumOn := TRUE;
            Crane$MagazinVacuumOff := FALSE;
            IF Crane$CraneSucked THEN
                Crane$_transit := TRUE;
                Crane$_state := Crane_states_t#Crane_Lift_At_Stamp2;
            END_IF

        Crane_states_t#TimeDelay:
            Crane$_transit := FALSE;
            Crane$TimeDelay_Timer$IN := TRUE;
            Crane$TimeDelay_Timer$PT := Crane$TimeDelay_Timer_Duration;
            IF Crane$TimeDelay_Timer$IN THEN
                Crane$TimeDelay_Timer$Q := (Crane$TimeDelay_Timer$ET = USINT#0);
                IF (Crane$TimeDelay_Timer$ET > USINT#0) THEN
                    Crane$TimeDelay_Timer$ET := (Crane$TimeDelay_Timer$ET - USINT#1);
                ELSE
                    Crane$TimeDelay_Timer$ET := USINT#0;
                END_IF
            ELSE
                Crane$TimeDelay_Timer$Q := FALSE;
                Crane$TimeDelay_Timer$ET := Crane$TimeDelay_Timer$PT;
            END_IF
            Crane$TimeDelay_Timer_interconnect := Crane$TimeDelay_Timer$Q;
            IF Crane$TimeDelay_Timer_interconnect THEN
                Crane$_transit := TRUE;
                Crane$_state := Crane_states_t#Interstep_3;
            END_IF

        Crane_states_t#Turn_Right:
            Crane$_transit := FALSE;
            Crane$CraneTurnClockwise := TRUE;
            Crane$CraneTurnCounterclockwise := FALSE;
            IF ((Crane$AnalogCranePosition > INT#24290) AND (Crane$AnalogCranePosition < INT#24390)) THEN
                Crane$_transit := TRUE;
                Crane$_state := Crane_states_t#Magazin_Stop;
            END_IF

        Crane_states_t#Turn_Right_Black:
            Crane$_transit := FALSE;
            Crane$CraneTurnClockwise := TRUE;
            Crane$CraneTurnCounterclockwise := FALSE;
            IF ((Crane$AnalogCranePosition > INT#24290) AND (Crane$AnalogCranePosition < INT#24390)) THEN
                Crane$_transit := TRUE;
                Crane$_state := Crane_states_t#Magazin_Stop_Black;
            END_IF

        Crane_states_t#Turn_Right_Final:
            Crane$_transit := FALSE;
            Crane$CraneTurnClockwise := TRUE;
            Crane$CraneTurnCounterclockwise := FALSE;
            Crane$AnalogCranePressure := INT#0;
            IF ((Crane$AnalogCranePosition > INT#24290) AND (Crane$AnalogCranePosition < INT#24390)) THEN
                Crane$_transit := TRUE;
                Crane$_state := Crane_states_t#Magazin_Stop_Final;
            END_IF

        Crane_states_t#pause:
            Crane$_transit := FALSE;
            Crane$Timer1$IN := Crane$CraneUp;
            Crane$Timer1$PT := Crane$Duration1;
            IF Crane$Timer1$IN THEN
                Crane$Timer1$Q := (Crane$Timer1$ET = USINT#0);
                IF (Crane$Timer1$ET > USINT#0) THEN
                    Crane$Timer1$ET := (Crane$Timer1$ET - USINT#1);
                ELSE
                    Crane$Timer1$ET := USINT#0;
                END_IF
            ELSE
                Crane$Timer1$Q := FALSE;
                Crane$Timer1$ET := Crane$Timer1$PT;
            END_IF
            Crane$interconnect := Crane$Timer1$Q;
            IF Crane$interconnect THEN
                Crane$_transit := TRUE;
                Crane$_state := Crane_states_t#Reset_interconnect;
            END_IF

        Crane_states_t#release:
            Crane$_transit := FALSE;
            Crane$MagazinVacuumOff := TRUE;
            Crane$MagazinVacuumOn := FALSE;
            IF TRUE THEN
                Crane$_transit := TRUE;
                Crane$_state := Crane_states_t#Crane_Lift_Conveyor;
            END_IF

        Crane_states_t#release2:
            Crane$_transit := FALSE;
            Crane$MagazinVacuumOff := TRUE;
            Crane$MagazinVacuumOn := FALSE;
            IF TRUE THEN
                Crane$_transit := TRUE;
                Crane$_state := Crane_states_t#Crane_Lift_Conveyor2;
            END_IF

        Crane_states_t#release_Black:
            Crane$_transit := FALSE;
            Crane$MagazinVacuumOn := FALSE;
            Crane$MagazinVacuumOff := TRUE;
            IF TRUE THEN
                Crane$_transit := TRUE;
                Crane$_state := Crane_states_t#Crane_Lift_Conveyor_Black;
            END_IF

        Crane_states_t#release_Workpiece:
            Crane$_transit := FALSE;
            Crane$MagazinVacuumOff := TRUE;
            Crane$MagazinVacuumOn := FALSE;
            IF TRUE THEN
                Crane$_transit := TRUE;
                Crane$_state := Crane_states_t#Crane_Go_Up;
            END_IF

        Crane_states_t#release_Workpiece_White:
            Crane$_transit := FALSE;
            Crane$MagazinVacuumOff := TRUE;
            Crane$MagazinVacuumOn := FALSE;
            IF TRUE THEN
                Crane$_transit := TRUE;
                Crane$_state := Crane_states_t#Crane_Go_Up_White;
            END_IF

            END_CASE
    CASE Stamp$_state OF
        Stamp_states_t#Green_Lamp:
            Stamp$_transit := FALSE;
            Stamp$StampGreenLamp := TRUE;
            Stamp$interconnectStampStartCommand := FALSE;
            IF TRUE THEN
                Stamp$_transit := TRUE;
                Stamp$_state := Stamp_states_t#Stamp_Init_1;
            END_IF

        Stamp_states_t#Init:
            Stamp$_transit := FALSE;
            IF TRUE THEN
                Stamp$_transit := TRUE;
                Stamp$_state := Stamp_states_t#Start_Stamp;
            END_IF

        Stamp_states_t#Interstep:
            Stamp$_transit := FALSE;
            Stamp$StartCommandStamp := TRUE;
            IF Stamp$StartVar THEN
                Stamp$_transit := TRUE;
                Stamp$_state := Stamp_states_t#Intertsep_2;
            END_IF

        Stamp_states_t#Intertsep_2:
            Stamp$_transit := FALSE;
            IF Stamp$StampSliderFilled THEN
                Stamp$_transit := TRUE;
                Stamp$_state := Stamp_states_t#Step0;
            END_IF

        Stamp_states_t#StampProcess:
            Stamp$_transit := FALSE;
            Stamp$StampSliderMovedIn := FALSE;
            Stamp$StampPusher := TRUE;
            IF Stamp$StampLowered THEN
                Stamp$_transit := TRUE;
                Stamp$_state := Stamp_states_t#Step1;
            END_IF

        Stamp_states_t#StampSliderBack:
            Stamp$_transit := FALSE;
            Stamp$StampSliderMovedIn := TRUE;
            Stamp$StampSliderMovedOut := FALSE;
            IF Stamp$StampSliderSensorMovedIn THEN
                Stamp$_transit := TRUE;
                Stamp$_state := Stamp_states_t#StampProcess;
            END_IF

        Stamp_states_t#StampSliderForward:
            Stamp$_transit := FALSE;
            Stamp$StampPusher := FALSE;
            Stamp$StampSliderMovedOut := TRUE;
            IF ((Stamp$StampLowered = FALSE) AND (Stamp$StampUp = TRUE)) THEN
                Stamp$interconnect := FALSE;
            END_IF
            Stamp$Timer$IN := FALSE;
            Stamp$Timer$PT := USINT#0;
            IF Stamp$Timer$IN THEN
                Stamp$Timer$Q := (Stamp$Timer$ET = USINT#0);
                IF (Stamp$Timer$ET > USINT#0) THEN
                    Stamp$Timer$ET := (Stamp$Timer$ET - USINT#1);
                ELSE
                    Stamp$Timer$ET := USINT#0;
                END_IF
            ELSE
                Stamp$Timer$Q := FALSE;
                Stamp$Timer$ET := Stamp$Timer$PT;
            END_IF
            IF Stamp$StampSliderMovedOut THEN
                Stamp$_transit := TRUE;
                Stamp$_state := Stamp_states_t#Step2;
            END_IF

        Stamp_states_t#Stamp_Init_1:
            Stamp$_transit := FALSE;
            Stamp$StampSliderMovedIn := TRUE;
            Stamp$StampSliderMovedOut := FALSE;
            IF Stamp$StampSliderSensorMovedIn THEN
                Stamp$_transit := TRUE;
                Stamp$_state := Stamp_states_t#Stamp_Init_2;
            END_IF

        Stamp_states_t#Stamp_Init_2:
            Stamp$_transit := FALSE;
            Stamp$StampSliderMovedIn := FALSE;
            Stamp$StampSliderMovedOut := TRUE;
            IF Stamp$StampSliderSensorMovedOut THEN
                Stamp$_transit := TRUE;
                Stamp$_state := Stamp_states_t#Stamp_Init_3;
            END_IF

        Stamp_states_t#Stamp_Init_3:
            Stamp$_transit := FALSE;
            Stamp$StampPusher := TRUE;
            IF Stamp$StampLowered THEN
                Stamp$_transit := TRUE;
                Stamp$_state := Stamp_states_t#Stamp_Init_4;
            END_IF

        Stamp_states_t#Stamp_Init_4:
            Stamp$_transit := FALSE;
            Stamp$StampPusher := FALSE;
            IF Stamp$StampUp THEN
                Stamp$_transit := TRUE;
                Stamp$_state := Stamp_states_t#Interstep;
            END_IF

        Stamp_states_t#Start_Stamp:
            Stamp$_transit := FALSE;
            Stamp$StampSliderMovedOut := FALSE;
            Stamp$StampSliderMovedIn := FALSE;
            Stamp$StampPusher := FALSE;
            Stamp$StampGreenLamp := FALSE;
            Stamp$StampPressure := FALSE;
            Stamp$StartCommandStamp := FALSE;
            IF (Stamp$StampStartButton = TRUE) THEN
                Stamp$interconnectStampStartCommand := TRUE;
            END_IF
            IF Stamp$interconnectStampStartCommand THEN
                Stamp$_transit := TRUE;
                Stamp$_state := Stamp_states_t#Green_Lamp;
            END_IF

        Stamp_states_t#Step0:
            Stamp$_transit := FALSE;
            IF Stamp$CraneUp THEN
                Stamp$_transit := TRUE;
                Stamp$_state := Stamp_states_t#StampSliderBack;
            END_IF

        Stamp_states_t#Step1:
            Stamp$_transit := FALSE;
            Stamp$Timer$IN := Stamp$StampLowered;
            Stamp$Timer$PT := USINT#0;
            IF Stamp$Timer$IN THEN
                Stamp$Timer$Q := (Stamp$Timer$ET = USINT#0);
                IF (Stamp$Timer$ET > USINT#0) THEN
                    Stamp$Timer$ET := (Stamp$Timer$ET - USINT#1);
                ELSE
                    Stamp$Timer$ET := USINT#0;
                END_IF
            ELSE
                Stamp$Timer$Q := FALSE;
                Stamp$Timer$ET := Stamp$Timer$PT;
            END_IF
            Stamp$interconnect := Stamp$Timer$Q;
            IF Stamp$interconnect THEN
                Stamp$_transit := TRUE;
                Stamp$_state := Stamp_states_t#StampSliderForward;
            END_IF

        Stamp_states_t#Step2:
            Stamp$_transit := FALSE;
            IF (((Stamp$AnalogCranePosition > INT#16160) AND (Stamp$AnalogCranePosition < INT#16260)) AND NOT Stamp$StampSliderFilled) THEN
                Stamp$_transit := TRUE;
                Stamp$_state := Stamp_states_t#Interstep;
            END_IF

            END_CASE
    CASE Conveyor$_state OF
        Conveyor_states_t#Conveyor_Init:
            Conveyor$_transit := FALSE;
            Conveyor$SorterConveyorTowardsStacker := TRUE;
            Conveyor$SorterConveyorTowardsCrane := FALSE;
            Conveyor$Timer_Conveyor_Test$IN := TRUE;
            Conveyor$Timer_Conveyor_Test$PT := Conveyor$Duration_Conveyor_Test;
            IF Conveyor$Timer_Conveyor_Test$IN THEN
                Conveyor$Timer_Conveyor_Test$Q := (Conveyor$Timer_Conveyor_Test$ET = USINT#0);
                IF (Conveyor$Timer_Conveyor_Test$ET > USINT#0) THEN
                    Conveyor$Timer_Conveyor_Test$ET := (Conveyor$Timer_Conveyor_Test$ET - USINT#1);
                ELSE
                    Conveyor$Timer_Conveyor_Test$ET := USINT#0;
                END_IF
            ELSE
                Conveyor$Timer_Conveyor_Test$Q := FALSE;
                Conveyor$Timer_Conveyor_Test$ET := Conveyor$Timer_Conveyor_Test$PT;
            END_IF
            Conveyor$interconnect_Conveyor_Test := Conveyor$Timer_Conveyor_Test$Q;
            IF Conveyor$interconnect_Conveyor_Test THEN
                Conveyor$_transit := TRUE;
                Conveyor$_state := Conveyor_states_t#Conveyor_init_2;
            END_IF

        Conveyor_states_t#Conveyor_Stop_Empty_Magazin:
            Conveyor$_transit := FALSE;
            Conveyor$SorterConveyorTowardsStacker := FALSE;
            Conveyor$SorterConveyorTowardsCrane := FALSE;
            Conveyor$interconnectConveyorStartCommand := FALSE;
            IF TRUE THEN
                Conveyor$_transit := TRUE;
                Conveyor$_state := Conveyor_states_t#Interstep;
            END_IF

        Conveyor_states_t#Conveyor_Towards_Stacker:
            Conveyor$_transit := FALSE;
            Conveyor$SorterConveyorTowardsStacker := TRUE;
            Conveyor$SorterConveyorTowardsCrane := FALSE;
            IF TRUE THEN
                Conveyor$_transit := TRUE;
                Conveyor$_state := Conveyor_states_t#Runtime_Conveyor;
            END_IF

        Conveyor_states_t#Conveyor_init_2:
            Conveyor$_transit := FALSE;
            Conveyor$SorterConveyorTowardsStacker := FALSE;
            Conveyor$SorterConveyorTowardsCrane := FALSE;
            Conveyor$interconnect_Conveyor_Test := FALSE;
            Conveyor$Timer_Conveyor_Test$IN := FALSE;
            Conveyor$Timer_Conveyor_Test$PT := USINT#0;
            IF Conveyor$Timer_Conveyor_Test$IN THEN
                Conveyor$Timer_Conveyor_Test$Q := (Conveyor$Timer_Conveyor_Test$ET = USINT#0);
                IF (Conveyor$Timer_Conveyor_Test$ET > USINT#0) THEN
                    Conveyor$Timer_Conveyor_Test$ET := (Conveyor$Timer_Conveyor_Test$ET - USINT#1);
                ELSE
                    Conveyor$Timer_Conveyor_Test$ET := USINT#0;
                END_IF
            ELSE
                Conveyor$Timer_Conveyor_Test$Q := FALSE;
                Conveyor$Timer_Conveyor_Test$ET := Conveyor$Timer_Conveyor_Test$PT;
            END_IF
            IF TRUE THEN
                Conveyor$_transit := TRUE;
                Conveyor$_state := Conveyor_states_t#Interstep;
            END_IF

        Conveyor_states_t#Conveyor_pause:
            Conveyor$_transit := FALSE;
            Conveyor$SorterConveyorTowardsStacker := FALSE;
            Conveyor$SorterConveyorTowardsCrane := FALSE;
            Conveyor$interconnect_Conveyor_Runtime := FALSE;
            Conveyor$Timer_Conveyor_Runtime$IN := FALSE;
            Conveyor$Timer_Conveyor_Runtime$PT := USINT#0;
            IF Conveyor$Timer_Conveyor_Runtime$IN THEN
                Conveyor$Timer_Conveyor_Runtime$Q := (Conveyor$Timer_Conveyor_Runtime$ET = USINT#0);
                IF (Conveyor$Timer_Conveyor_Runtime$ET > USINT#0) THEN
                    Conveyor$Timer_Conveyor_Runtime$ET := (Conveyor$Timer_Conveyor_Runtime$ET - USINT#1);
                ELSE
                    Conveyor$Timer_Conveyor_Runtime$ET := USINT#0;
                END_IF
            ELSE
                Conveyor$Timer_Conveyor_Runtime$Q := FALSE;
                Conveyor$Timer_Conveyor_Runtime$ET := Conveyor$Timer_Conveyor_Runtime$PT;
            END_IF
            IF TRUE THEN
                Conveyor$_transit := TRUE;
                Conveyor$_state := Conveyor_states_t#Interstep;
            END_IF

        Conveyor_states_t#Green_Lamp:
            Conveyor$_transit := FALSE;
            Conveyor$SorterGreenLampConveyor := TRUE;
            Conveyor$interconnectConveyorStartCommand := FALSE;
            IF TRUE THEN
                Conveyor$_transit := TRUE;
                Conveyor$_state := Conveyor_states_t#Conveyor_Init;
            END_IF

        Conveyor_states_t#Init:
            Conveyor$_transit := FALSE;
            IF TRUE THEN
                Conveyor$_transit := TRUE;
                Conveyor$_state := Conveyor_states_t#Start_Conveyor;
            END_IF

        Conveyor_states_t#Interstep:
            Conveyor$_transit := FALSE;
            Conveyor$StartCommandConveyor := TRUE;
            IF Conveyor$StartVar THEN
                Conveyor$_transit := TRUE;
                Conveyor$_state := Conveyor_states_t#Step0;
            END_IF

        Conveyor_states_t#Runtime_Conveyor:
            Conveyor$_transit := FALSE;
            Conveyor$Timer_Conveyor_Runtime$IN := TRUE;
            Conveyor$Timer_Conveyor_Runtime$PT := Conveyor$Duration_Conveyor_Runtime;
            IF Conveyor$Timer_Conveyor_Runtime$IN THEN
                Conveyor$Timer_Conveyor_Runtime$Q := (Conveyor$Timer_Conveyor_Runtime$ET = USINT#0);
                IF (Conveyor$Timer_Conveyor_Runtime$ET > USINT#0) THEN
                    Conveyor$Timer_Conveyor_Runtime$ET := (Conveyor$Timer_Conveyor_Runtime$ET - USINT#1);
                ELSE
                    Conveyor$Timer_Conveyor_Runtime$ET := USINT#0;
                END_IF
            ELSE
                Conveyor$Timer_Conveyor_Runtime$Q := FALSE;
                Conveyor$Timer_Conveyor_Runtime$ET := Conveyor$Timer_Conveyor_Runtime$PT;
            END_IF
            Conveyor$interconnect_Conveyor_Runtime := Conveyor$Timer_Conveyor_Runtime$Q;
            IF Conveyor$interconnect_Conveyor_Runtime THEN
                Conveyor$_transit := TRUE;
                Conveyor$_state := Conveyor_states_t#Conveyor_pause;
            END_IF

        Conveyor_states_t#Start_Conveyor:
            Conveyor$_transit := FALSE;
            Conveyor$interconnectConveyorTerminationCommand := FALSE;
            Conveyor$SorterConveyorTowardsStacker := FALSE;
            Conveyor$SorterConveyorTowardsCrane := FALSE;
            Conveyor$SorterGreenLampConveyor := FALSE;
            Conveyor$interconnect_Conveyor_Runtime := FALSE;
            Conveyor$interconnect_Conveyor_Test := FALSE;
            Conveyor$Timer_Conveyor_Test$IN := FALSE;
            Conveyor$Timer_Conveyor_Test$PT := USINT#0;
            IF Conveyor$Timer_Conveyor_Test$IN THEN
                Conveyor$Timer_Conveyor_Test$Q := (Conveyor$Timer_Conveyor_Test$ET = USINT#0);
                IF (Conveyor$Timer_Conveyor_Test$ET > USINT#0) THEN
                    Conveyor$Timer_Conveyor_Test$ET := (Conveyor$Timer_Conveyor_Test$ET - USINT#1);
                ELSE
                    Conveyor$Timer_Conveyor_Test$ET := USINT#0;
                END_IF
            ELSE
                Conveyor$Timer_Conveyor_Test$Q := FALSE;
                Conveyor$Timer_Conveyor_Test$ET := Conveyor$Timer_Conveyor_Test$PT;
            END_IF
            Conveyor$Timer_Conveyor_Runtime$IN := FALSE;
            Conveyor$Timer_Conveyor_Runtime$PT := USINT#0;
            IF Conveyor$Timer_Conveyor_Runtime$IN THEN
                Conveyor$Timer_Conveyor_Runtime$Q := (Conveyor$Timer_Conveyor_Runtime$ET = USINT#0);
                IF (Conveyor$Timer_Conveyor_Runtime$ET > USINT#0) THEN
                    Conveyor$Timer_Conveyor_Runtime$ET := (Conveyor$Timer_Conveyor_Runtime$ET - USINT#1);
                ELSE
                    Conveyor$Timer_Conveyor_Runtime$ET := USINT#0;
                END_IF
            ELSE
                Conveyor$Timer_Conveyor_Runtime$Q := FALSE;
                Conveyor$Timer_Conveyor_Runtime$ET := Conveyor$Timer_Conveyor_Runtime$PT;
            END_IF
            Conveyor$StartVar := FALSE;
            Conveyor$StartCommandConveyor := FALSE;
            IF (Conveyor$SorterStartButton = TRUE) THEN
                Conveyor$interconnectConveyorStartCommand := TRUE;
            END_IF
            IF Conveyor$interconnectConveyorStartCommand THEN
                Conveyor$_transit := TRUE;
                Conveyor$_state := Conveyor_states_t#Green_Lamp;
            END_IF

        Conveyor_states_t#Step0:
            Conveyor$_transit := FALSE;
            IF Conveyor$SorterLightbarrierCraneInterface THEN
                Conveyor$_transit := TRUE;
                Conveyor$_state := Conveyor_states_t#Conveyor_Towards_Stacker;
            ELSEIF NOT Conveyor$SorterLightbarrierCraneInterface THEN
                Conveyor$_transit := TRUE;
                Conveyor$_state := Conveyor_states_t#Conveyor_Stop_Empty_Magazin;
            END_IF

            END_CASE
    CASE Pusher$_state OF
        Pusher_states_t#Check_For_Black:
            Pusher$_transit := FALSE;
            IF ((Pusher$Slide2_black = INT#1) AND (Pusher$Priority_Var_Black = INT#2)) THEN
                Pusher$_transit := TRUE;
                Pusher$_state := Pusher_states_t#Second_Slide_black_workpieces;
            ELSEIF ((Pusher$Slide3_black = INT#1) AND (Pusher$Priority_Var_Black = INT#3)) THEN
                Pusher$_transit := TRUE;
                Pusher$_state := Pusher_states_t#Third_Slide_black_workpieces;
            ELSEIF ((Pusher$Slide1_black = INT#1) AND (Pusher$Priority_Var_Black = INT#1)) THEN
                Pusher$_transit := TRUE;
                Pusher$_state := Pusher_states_t#First_Slide_black_workpieces;
            END_IF

        Pusher_states_t#Check_For_Metal:
            Pusher$_transit := FALSE;
            IF ((Pusher$Slide3_metal = INT#1) AND (Pusher$Priority_Var_Metal = INT#3)) THEN
                Pusher$_transit := TRUE;
                Pusher$_state := Pusher_states_t#Third_Slide_metal_workpieces;
            ELSEIF ((Pusher$Slide2_metal = INT#1) AND (Pusher$Priority_Var_Metal = INT#2)) THEN
                Pusher$_transit := TRUE;
                Pusher$_state := Pusher_states_t#Second_Slide_metal_workpieces;
            ELSEIF ((Pusher$Slide1_metal = INT#1) AND (Pusher$Priority_Var_Metal = INT#1)) THEN
                Pusher$_transit := TRUE;
                Pusher$_state := Pusher_states_t#First_Slide_metal_workpieces;
            END_IF

        Pusher_states_t#Check_For_White:
            Pusher$_transit := FALSE;
            IF ((Pusher$Slide1_white = INT#1) AND (Pusher$Priority_Var_White = INT#1)) THEN
                Pusher$_transit := TRUE;
                Pusher$_state := Pusher_states_t#First_Slide_white_workpieces;
            ELSEIF ((Pusher$Slide3_white = INT#1) AND (Pusher$Priority_Var_White = INT#3)) THEN
                Pusher$_transit := TRUE;
                Pusher$_state := Pusher_states_t#Third_Slide_white_workpieces;
            ELSEIF ((Pusher$Slide2_white = INT#1) AND (Pusher$Priority_Var_White = INT#2)) THEN
                Pusher$_transit := TRUE;
                Pusher$_state := Pusher_states_t#Second_Slide_white_workpieces;
            END_IF

        Pusher_states_t#First_Slide_Timer_Black:
            Pusher$_transit := FALSE;
            IF (Pusher$SorterLightnesssensorCraneInterfaceInverse = TRUE) THEN
                Pusher$Timer_Slide1_Black$IN := Pusher$SorterLightnesssensorCraneInterfaceInverse;
                Pusher$Timer_Slide1_Black$PT := Pusher$Duration_Slide1_Black;
                IF Pusher$Timer_Slide1_Black$IN THEN
                    Pusher$Timer_Slide1_Black$Q := (Pusher$Timer_Slide1_Black$ET = USINT#0);
                    IF (Pusher$Timer_Slide1_Black$ET > USINT#0) THEN
                        Pusher$Timer_Slide1_Black$ET := (Pusher$Timer_Slide1_Black$ET - USINT#1);
                    ELSE
                        Pusher$Timer_Slide1_Black$ET := USINT#0;
                    END_IF
                ELSE
                    Pusher$Timer_Slide1_Black$Q := FALSE;
                    Pusher$Timer_Slide1_Black$ET := Pusher$Timer_Slide1_Black$PT;
                END_IF
                Pusher$interconnect_Slide1_Black := Pusher$Timer_Slide1_Black$Q;
            END_IF
            IF Pusher$interconnect_Slide1_Black THEN
                Pusher$_transit := TRUE;
                Pusher$_state := Pusher_states_t#PusherY1_Move_Out_Black;
            END_IF

        Pusher_states_t#First_Slide_Timer_Metal:
            Pusher$_transit := FALSE;
            Pusher$Timer_Slide1_Metal$IN := TRUE;
            Pusher$Timer_Slide1_Metal$PT := Pusher$Duration_Slide1_Metal;
            IF Pusher$Timer_Slide1_Metal$IN THEN
                Pusher$Timer_Slide1_Metal$Q := (Pusher$Timer_Slide1_Metal$ET = USINT#0);
                IF (Pusher$Timer_Slide1_Metal$ET > USINT#0) THEN
                    Pusher$Timer_Slide1_Metal$ET := (Pusher$Timer_Slide1_Metal$ET - USINT#1);
                ELSE
                    Pusher$Timer_Slide1_Metal$ET := USINT#0;
                END_IF
            ELSE
                Pusher$Timer_Slide1_Metal$Q := FALSE;
                Pusher$Timer_Slide1_Metal$ET := Pusher$Timer_Slide1_Metal$PT;
            END_IF
            Pusher$interconnect_Slide1_Metal := Pusher$Timer_Slide1_Metal$Q;
            IF Pusher$interconnect_Slide1_Metal THEN
                Pusher$_transit := TRUE;
                Pusher$_state := Pusher_states_t#PusherY1_Move_Out_Metal;
            END_IF

        Pusher_states_t#First_Slide_Timer_White:
            Pusher$_transit := FALSE;
            Pusher$Timer_Slide1_White$IN := TRUE;
            Pusher$Timer_Slide1_White$PT := Pusher$Duration_Slide1_White;
            IF Pusher$Timer_Slide1_White$IN THEN
                Pusher$Timer_Slide1_White$Q := (Pusher$Timer_Slide1_White$ET = USINT#0);
                IF (Pusher$Timer_Slide1_White$ET > USINT#0) THEN
                    Pusher$Timer_Slide1_White$ET := (Pusher$Timer_Slide1_White$ET - USINT#1);
                ELSE
                    Pusher$Timer_Slide1_White$ET := USINT#0;
                END_IF
            ELSE
                Pusher$Timer_Slide1_White$Q := FALSE;
                Pusher$Timer_Slide1_White$ET := Pusher$Timer_Slide1_White$PT;
            END_IF
            Pusher$interconnect_Slide1_White := Pusher$Timer_Slide1_White$Q;
            IF Pusher$interconnect_Slide1_White THEN
                Pusher$_transit := TRUE;
                Pusher$_state := Pusher_states_t#PusherY1_Move_Out_White;
            END_IF

        Pusher_states_t#First_Slide_black_workpieces:
            Pusher$_transit := FALSE;
            IF TRUE THEN
                Pusher$_transit := TRUE;
                Pusher$_state := Pusher_states_t#First_Slide_Timer_Black;
            END_IF

        Pusher_states_t#First_Slide_metal_workpieces:
            Pusher$_transit := FALSE;
            IF TRUE THEN
                Pusher$_transit := TRUE;
                Pusher$_state := Pusher_states_t#First_Slide_Timer_Metal;
            END_IF

        Pusher_states_t#First_Slide_white_workpieces:
            Pusher$_transit := FALSE;
            IF TRUE THEN
                Pusher$_transit := TRUE;
                Pusher$_state := Pusher_states_t#First_Slide_Timer_White;
            END_IF

        Pusher_states_t#Init:
            Pusher$_transit := FALSE;
            IF Pusher$StartVar THEN
                Pusher$_transit := TRUE;
                Pusher$_state := Pusher_states_t#Interstep;
            END_IF

        Pusher_states_t#Interstep:
            Pusher$_transit := FALSE;
            Pusher$PusherY1 := FALSE;
            Pusher$PusherY2 := FALSE;
            Pusher$interconnect2 := FALSE;
            Pusher$interconnect3 := FALSE;
            Pusher$StartVar := FALSE;
            Pusher$interconnect_Slide1_Black := FALSE;
            Pusher$interconnect_Slide2_Black := FALSE;
            Pusher$interconnect_Slide1_White := FALSE;
            Pusher$interconnect_Slide2_White := FALSE;
            Pusher$interconnect_Slide1_Metal := FALSE;
            Pusher$interconnect_Slide2_Metal := FALSE;
            IF TRUE THEN
                Pusher$_transit := TRUE;
                Pusher$_state := Pusher_states_t#Interstep_2;
            END_IF

        Pusher_states_t#Interstep_2:
            Pusher$_transit := FALSE;
            IF ((Pusher$SorterLightnessSensorPusher1 AND Pusher$SorterCapacitiveSensorPusher1) AND (Pusher$Priority_Var_Metal > INT#0)) THEN
                Pusher$_transit := TRUE;
                Pusher$_state := Pusher_states_t#Check_For_Metal;
            ELSEIF ((NOT Pusher$SorterLightnesssensorCraneInterfaceInverse AND Pusher$SorterLightbarrierCraneInterface) AND (Pusher$Priority_Var_Black > INT#0)) THEN
                Pusher$_transit := TRUE;
                Pusher$_state := Pusher_states_t#Check_For_Black;
            ELSEIF ((Pusher$SorterLightnessSensorPusher1 AND NOT Pusher$SorterCapacitiveSensorPusher1) AND (Pusher$Priority_Var_White > INT#0)) THEN
                Pusher$_transit := TRUE;
                Pusher$_state := Pusher_states_t#Check_For_White;
            END_IF

        Pusher_states_t#PusherY1_Move_In_Black:
            Pusher$_transit := FALSE;
            IF ((Pusher$SorterPusher1MovedOut = TRUE) AND (Pusher$SorterPusher1MovedIn = FALSE)) THEN
                Pusher$PusherY1 := FALSE;
            END_IF
            IF Pusher$SorterPusher1MovedIn THEN
                Pusher$_transit := TRUE;
                Pusher$_state := Pusher_states_t#Reset_interconnect_Slide1_Black;
            END_IF

        Pusher_states_t#PusherY1_Move_In_Metal:
            Pusher$_transit := FALSE;
            IF ((Pusher$SorterPusher1MovedOut = TRUE) AND (Pusher$SorterPusher1MovedIn = FALSE)) THEN
                Pusher$PusherY1 := FALSE;
            END_IF
            IF Pusher$SorterPusher1MovedIn THEN
                Pusher$_transit := TRUE;
                Pusher$_state := Pusher_states_t#Reset_interconnect_Slide1_Metal;
            END_IF

        Pusher_states_t#PusherY1_Move_In_White:
            Pusher$_transit := FALSE;
            IF ((Pusher$SorterPusher1MovedOut = TRUE) AND (Pusher$SorterPusher1MovedIn = FALSE)) THEN
                Pusher$PusherY1 := FALSE;
            END_IF
            IF Pusher$SorterPusher1MovedIn THEN
                Pusher$_transit := TRUE;
                Pusher$_state := Pusher_states_t#Reset_interconnect_Slide1_White;
            END_IF

        Pusher_states_t#PusherY1_Move_Out_Black:
            Pusher$_transit := FALSE;
            IF ((Pusher$SorterPusher1MovedOut = FALSE) AND (Pusher$SorterPusher1MovedIn = TRUE)) THEN
                Pusher$PusherY1 := TRUE;
            END_IF
            IF Pusher$SorterPusher1MovedOut THEN
                Pusher$_transit := TRUE;
                Pusher$_state := Pusher_states_t#Wait_Y1_Black;
            END_IF

        Pusher_states_t#PusherY1_Move_Out_Metal:
            Pusher$_transit := FALSE;
            IF ((Pusher$SorterPusher1MovedOut = FALSE) AND (Pusher$SorterPusher1MovedIn = TRUE)) THEN
                Pusher$PusherY1 := TRUE;
            END_IF
            IF Pusher$SorterPusher1MovedOut THEN
                Pusher$_transit := TRUE;
                Pusher$_state := Pusher_states_t#Wait_Y1_Metal;
            END_IF

        Pusher_states_t#PusherY1_Move_Out_White:
            Pusher$_transit := FALSE;
            IF ((Pusher$SorterPusher1MovedOut = FALSE) AND (Pusher$SorterPusher1MovedIn = TRUE)) THEN
                Pusher$PusherY1 := TRUE;
            END_IF
            IF Pusher$SorterPusher1MovedOut THEN
                Pusher$_transit := TRUE;
                Pusher$_state := Pusher_states_t#Wait_Y1_White;
            END_IF

        Pusher_states_t#PusherY2_Move_In_Black:
            Pusher$_transit := FALSE;
            IF ((Pusher$SorterPusher2MovedOut = TRUE) AND (Pusher$SorterPusher2MovedIn = FALSE)) THEN
                Pusher$PusherY2 := FALSE;
            END_IF
            IF Pusher$SorterPusher2MovedIn THEN
                Pusher$_transit := TRUE;
                Pusher$_state := Pusher_states_t#Reset_interconnect_Slide2_Black;
            END_IF

        Pusher_states_t#PusherY2_Move_In_Metal:
            Pusher$_transit := FALSE;
            IF ((Pusher$SorterPusher2MovedOut = TRUE) AND (Pusher$SorterPusher2MovedIn = FALSE)) THEN
                Pusher$PusherY2 := FALSE;
            END_IF
            IF Pusher$SorterPusher2MovedIn THEN
                Pusher$_transit := TRUE;
                Pusher$_state := Pusher_states_t#Reset_interconnect_Slide2_Metal;
            END_IF

        Pusher_states_t#PusherY2_Move_In_White:
            Pusher$_transit := FALSE;
            IF ((Pusher$SorterPusher2MovedOut = TRUE) AND (Pusher$SorterPusher2MovedIn = FALSE)) THEN
                Pusher$PusherY2 := FALSE;
            END_IF
            IF Pusher$SorterPusher2MovedIn THEN
                Pusher$_transit := TRUE;
                Pusher$_state := Pusher_states_t#Reset_interconnect_Slide2_White;
            END_IF

        Pusher_states_t#PusherY2_Move_Out_Black:
            Pusher$_transit := FALSE;
            IF ((Pusher$SorterPusher2MovedOut = FALSE) AND (Pusher$SorterPusher2MovedIn = TRUE)) THEN
                Pusher$PusherY2 := TRUE;
            END_IF
            IF Pusher$SorterPusher2MovedOut THEN
                Pusher$_transit := TRUE;
                Pusher$_state := Pusher_states_t#Wait_Y2_Black;
            END_IF

        Pusher_states_t#PusherY2_Move_Out_Metal:
            Pusher$_transit := FALSE;
            IF ((Pusher$SorterPusher2MovedOut = FALSE) AND (Pusher$SorterPusher2MovedIn = TRUE)) THEN
                Pusher$PusherY2 := TRUE;
            END_IF
            IF Pusher$SorterPusher2MovedOut THEN
                Pusher$_transit := TRUE;
                Pusher$_state := Pusher_states_t#Wait_Y2_Metal;
            END_IF

        Pusher_states_t#PusherY2_Move_Out_White:
            Pusher$_transit := FALSE;
            IF ((Pusher$SorterPusher2MovedOut = FALSE) AND (Pusher$SorterPusher2MovedIn = TRUE)) THEN
                Pusher$PusherY2 := TRUE;
            END_IF
            IF Pusher$SorterPusher2MovedOut THEN
                Pusher$_transit := TRUE;
                Pusher$_state := Pusher_states_t#Wait_Y2_White;
            END_IF

        Pusher_states_t#Reset_interconnect3:
            Pusher$_transit := FALSE;
            Pusher$interconnect2 := FALSE;
            Pusher$Timer2$IN := FALSE;
            Pusher$Timer2$PT := USINT#0;
            IF Pusher$Timer2$IN THEN
                Pusher$Timer2$Q := (Pusher$Timer2$ET = USINT#0);
                IF (Pusher$Timer2$ET > USINT#0) THEN
                    Pusher$Timer2$ET := (Pusher$Timer2$ET - USINT#1);
                ELSE
                    Pusher$Timer2$ET := USINT#0;
                END_IF
            ELSE
                Pusher$Timer2$Q := FALSE;
                Pusher$Timer2$ET := Pusher$Timer2$PT;
            END_IF
            Pusher$Slide3_black := (Pusher$Slide3_black - INT#1);
            Pusher$Priority_Var_Black := (Pusher$Priority_Var_Black - INT#1);
            IF TRUE THEN
                Pusher$_transit := TRUE;
                Pusher$_state := Pusher_states_t#Interstep_2;
            END_IF

        Pusher_states_t#Reset_interconnect_Slide1_Black:
            Pusher$_transit := FALSE;
            Pusher$interconnect3 := FALSE;
            Pusher$Timer3$IN := FALSE;
            Pusher$Timer3$PT := USINT#0;
            IF Pusher$Timer3$IN THEN
                Pusher$Timer3$Q := (Pusher$Timer3$ET = USINT#0);
                IF (Pusher$Timer3$ET > USINT#0) THEN
                    Pusher$Timer3$ET := (Pusher$Timer3$ET - USINT#1);
                ELSE
                    Pusher$Timer3$ET := USINT#0;
                END_IF
            ELSE
                Pusher$Timer3$Q := FALSE;
                Pusher$Timer3$ET := Pusher$Timer3$PT;
            END_IF
            Pusher$interconnect_Slide1_Black := FALSE;
            Pusher$Timer_Slide1_Black$IN := FALSE;
            Pusher$Timer_Slide1_Black$PT := USINT#0;
            IF Pusher$Timer_Slide1_Black$IN THEN
                Pusher$Timer_Slide1_Black$Q := (Pusher$Timer_Slide1_Black$ET = USINT#0);
                IF (Pusher$Timer_Slide1_Black$ET > USINT#0) THEN
                    Pusher$Timer_Slide1_Black$ET := (Pusher$Timer_Slide1_Black$ET - USINT#1);
                ELSE
                    Pusher$Timer_Slide1_Black$ET := USINT#0;
                END_IF
            ELSE
                Pusher$Timer_Slide1_Black$Q := FALSE;
                Pusher$Timer_Slide1_Black$ET := Pusher$Timer_Slide1_Black$PT;
            END_IF
            Pusher$Slide1_black := (Pusher$Slide1_black - INT#1);
            Pusher$Priority_Var_Black := (Pusher$Priority_Var_Black - INT#1);
            IF TRUE THEN
                Pusher$_transit := TRUE;
                Pusher$_state := Pusher_states_t#Interstep_2;
            END_IF

        Pusher_states_t#Reset_interconnect_Slide1_Metal:
            Pusher$_transit := FALSE;
            Pusher$interconnect3 := FALSE;
            Pusher$Timer3$IN := FALSE;
            Pusher$Timer3$PT := USINT#0;
            IF Pusher$Timer3$IN THEN
                Pusher$Timer3$Q := (Pusher$Timer3$ET = USINT#0);
                IF (Pusher$Timer3$ET > USINT#0) THEN
                    Pusher$Timer3$ET := (Pusher$Timer3$ET - USINT#1);
                ELSE
                    Pusher$Timer3$ET := USINT#0;
                END_IF
            ELSE
                Pusher$Timer3$Q := FALSE;
                Pusher$Timer3$ET := Pusher$Timer3$PT;
            END_IF
            Pusher$interconnect_Slide1_Metal := FALSE;
            Pusher$Timer_Slide1_Metal$IN := FALSE;
            Pusher$Timer_Slide1_Metal$PT := USINT#0;
            IF Pusher$Timer_Slide1_Metal$IN THEN
                Pusher$Timer_Slide1_Metal$Q := (Pusher$Timer_Slide1_Metal$ET = USINT#0);
                IF (Pusher$Timer_Slide1_Metal$ET > USINT#0) THEN
                    Pusher$Timer_Slide1_Metal$ET := (Pusher$Timer_Slide1_Metal$ET - USINT#1);
                ELSE
                    Pusher$Timer_Slide1_Metal$ET := USINT#0;
                END_IF
            ELSE
                Pusher$Timer_Slide1_Metal$Q := FALSE;
                Pusher$Timer_Slide1_Metal$ET := Pusher$Timer_Slide1_Metal$PT;
            END_IF
            Pusher$Slide1_metal := (Pusher$Slide1_metal - INT#1);
            Pusher$Priority_Var_Metal := (Pusher$Priority_Var_Metal - INT#1);
            IF TRUE THEN
                Pusher$_transit := TRUE;
                Pusher$_state := Pusher_states_t#Interstep_2;
            END_IF

        Pusher_states_t#Reset_interconnect_Slide1_White:
            Pusher$_transit := FALSE;
            Pusher$interconnect3 := FALSE;
            Pusher$Timer3$IN := FALSE;
            Pusher$Timer3$PT := USINT#0;
            IF Pusher$Timer3$IN THEN
                Pusher$Timer3$Q := (Pusher$Timer3$ET = USINT#0);
                IF (Pusher$Timer3$ET > USINT#0) THEN
                    Pusher$Timer3$ET := (Pusher$Timer3$ET - USINT#1);
                ELSE
                    Pusher$Timer3$ET := USINT#0;
                END_IF
            ELSE
                Pusher$Timer3$Q := FALSE;
                Pusher$Timer3$ET := Pusher$Timer3$PT;
            END_IF
            Pusher$interconnect_Slide1_White := FALSE;
            Pusher$Timer_Slide1_White$IN := FALSE;
            Pusher$Timer_Slide1_White$PT := USINT#0;
            IF Pusher$Timer_Slide1_White$IN THEN
                Pusher$Timer_Slide1_White$Q := (Pusher$Timer_Slide1_White$ET = USINT#0);
                IF (Pusher$Timer_Slide1_White$ET > USINT#0) THEN
                    Pusher$Timer_Slide1_White$ET := (Pusher$Timer_Slide1_White$ET - USINT#1);
                ELSE
                    Pusher$Timer_Slide1_White$ET := USINT#0;
                END_IF
            ELSE
                Pusher$Timer_Slide1_White$Q := FALSE;
                Pusher$Timer_Slide1_White$ET := Pusher$Timer_Slide1_White$PT;
            END_IF
            Pusher$Slide1_white := (Pusher$Slide1_white - INT#1);
            Pusher$Priority_Var_White := (Pusher$Priority_Var_White - INT#1);
            IF TRUE THEN
                Pusher$_transit := TRUE;
                Pusher$_state := Pusher_states_t#Interstep_2;
            END_IF

        Pusher_states_t#Reset_interconnect_Slide2_Black:
            Pusher$_transit := FALSE;
            Pusher$interconnect3 := FALSE;
            Pusher$Timer3$IN := FALSE;
            Pusher$Timer3$PT := USINT#0;
            IF Pusher$Timer3$IN THEN
                Pusher$Timer3$Q := (Pusher$Timer3$ET = USINT#0);
                IF (Pusher$Timer3$ET > USINT#0) THEN
                    Pusher$Timer3$ET := (Pusher$Timer3$ET - USINT#1);
                ELSE
                    Pusher$Timer3$ET := USINT#0;
                END_IF
            ELSE
                Pusher$Timer3$Q := FALSE;
                Pusher$Timer3$ET := Pusher$Timer3$PT;
            END_IF
            Pusher$interconnect_Slide2_Black := FALSE;
            Pusher$Timer_Slide2_Black$IN := FALSE;
            Pusher$Timer_Slide2_Black$PT := USINT#0;
            IF Pusher$Timer_Slide2_Black$IN THEN
                Pusher$Timer_Slide2_Black$Q := (Pusher$Timer_Slide2_Black$ET = USINT#0);
                IF (Pusher$Timer_Slide2_Black$ET > USINT#0) THEN
                    Pusher$Timer_Slide2_Black$ET := (Pusher$Timer_Slide2_Black$ET - USINT#1);
                ELSE
                    Pusher$Timer_Slide2_Black$ET := USINT#0;
                END_IF
            ELSE
                Pusher$Timer_Slide2_Black$Q := FALSE;
                Pusher$Timer_Slide2_Black$ET := Pusher$Timer_Slide2_Black$PT;
            END_IF
            Pusher$Slide2_black := (Pusher$Slide2_black - INT#1);
            Pusher$Priority_Var_Black := (Pusher$Priority_Var_Black - INT#1);
            IF TRUE THEN
                Pusher$_transit := TRUE;
                Pusher$_state := Pusher_states_t#Interstep_2;
            END_IF

        Pusher_states_t#Reset_interconnect_Slide2_Metal:
            Pusher$_transit := FALSE;
            Pusher$interconnect3 := FALSE;
            Pusher$Timer3$IN := FALSE;
            Pusher$Timer3$PT := USINT#0;
            IF Pusher$Timer3$IN THEN
                Pusher$Timer3$Q := (Pusher$Timer3$ET = USINT#0);
                IF (Pusher$Timer3$ET > USINT#0) THEN
                    Pusher$Timer3$ET := (Pusher$Timer3$ET - USINT#1);
                ELSE
                    Pusher$Timer3$ET := USINT#0;
                END_IF
            ELSE
                Pusher$Timer3$Q := FALSE;
                Pusher$Timer3$ET := Pusher$Timer3$PT;
            END_IF
            Pusher$interconnect_Slide2_Metal := FALSE;
            Pusher$Timer_Slide2_Metal$IN := FALSE;
            Pusher$Timer_Slide2_Metal$PT := USINT#0;
            IF Pusher$Timer_Slide2_Metal$IN THEN
                Pusher$Timer_Slide2_Metal$Q := (Pusher$Timer_Slide2_Metal$ET = USINT#0);
                IF (Pusher$Timer_Slide2_Metal$ET > USINT#0) THEN
                    Pusher$Timer_Slide2_Metal$ET := (Pusher$Timer_Slide2_Metal$ET - USINT#1);
                ELSE
                    Pusher$Timer_Slide2_Metal$ET := USINT#0;
                END_IF
            ELSE
                Pusher$Timer_Slide2_Metal$Q := FALSE;
                Pusher$Timer_Slide2_Metal$ET := Pusher$Timer_Slide2_Metal$PT;
            END_IF
            Pusher$Slide2_metal := (Pusher$Slide2_metal - INT#1);
            Pusher$Priority_Var_Metal := (Pusher$Priority_Var_Metal - INT#1);
            IF TRUE THEN
                Pusher$_transit := TRUE;
                Pusher$_state := Pusher_states_t#Interstep_2;
            END_IF

        Pusher_states_t#Reset_interconnect_Slide2_White:
            Pusher$_transit := FALSE;
            Pusher$interconnect3 := FALSE;
            Pusher$Timer3$IN := FALSE;
            Pusher$Timer3$PT := USINT#0;
            IF Pusher$Timer3$IN THEN
                Pusher$Timer3$Q := (Pusher$Timer3$ET = USINT#0);
                IF (Pusher$Timer3$ET > USINT#0) THEN
                    Pusher$Timer3$ET := (Pusher$Timer3$ET - USINT#1);
                ELSE
                    Pusher$Timer3$ET := USINT#0;
                END_IF
            ELSE
                Pusher$Timer3$Q := FALSE;
                Pusher$Timer3$ET := Pusher$Timer3$PT;
            END_IF
            Pusher$interconnect_Slide2_White := FALSE;
            Pusher$Timer_Slide2_White$IN := FALSE;
            Pusher$Timer_Slide2_White$PT := USINT#0;
            IF Pusher$Timer_Slide2_White$IN THEN
                Pusher$Timer_Slide2_White$Q := (Pusher$Timer_Slide2_White$ET = USINT#0);
                IF (Pusher$Timer_Slide2_White$ET > USINT#0) THEN
                    Pusher$Timer_Slide2_White$ET := (Pusher$Timer_Slide2_White$ET - USINT#1);
                ELSE
                    Pusher$Timer_Slide2_White$ET := USINT#0;
                END_IF
            ELSE
                Pusher$Timer_Slide2_White$Q := FALSE;
                Pusher$Timer_Slide2_White$ET := Pusher$Timer_Slide2_White$PT;
            END_IF
            Pusher$Slide2_white := (Pusher$Slide2_white - INT#1);
            Pusher$Priority_Var_White := (Pusher$Priority_Var_White - INT#1);
            IF TRUE THEN
                Pusher$_transit := TRUE;
                Pusher$_state := Pusher_states_t#Interstep_2;
            END_IF

        Pusher_states_t#Reset_interconnect_Slide3_Metal:
            Pusher$_transit := FALSE;
            Pusher$interconnect3 := FALSE;
            Pusher$Timer3$IN := FALSE;
            Pusher$Timer3$PT := USINT#0;
            IF Pusher$Timer3$IN THEN
                Pusher$Timer3$Q := (Pusher$Timer3$ET = USINT#0);
                IF (Pusher$Timer3$ET > USINT#0) THEN
                    Pusher$Timer3$ET := (Pusher$Timer3$ET - USINT#1);
                ELSE
                    Pusher$Timer3$ET := USINT#0;
                END_IF
            ELSE
                Pusher$Timer3$Q := FALSE;
                Pusher$Timer3$ET := Pusher$Timer3$PT;
            END_IF
            Pusher$Slide3_metal := (Pusher$Slide3_metal - INT#1);
            Pusher$Priority_Var_Metal := (Pusher$Priority_Var_Metal - INT#1);
            IF TRUE THEN
                Pusher$_transit := TRUE;
                Pusher$_state := Pusher_states_t#Interstep_2;
            END_IF

        Pusher_states_t#Reset_interconnect_Slide3_White:
            Pusher$_transit := FALSE;
            Pusher$interconnect3 := FALSE;
            Pusher$Timer3$IN := FALSE;
            Pusher$Timer3$PT := USINT#0;
            IF Pusher$Timer3$IN THEN
                Pusher$Timer3$Q := (Pusher$Timer3$ET = USINT#0);
                IF (Pusher$Timer3$ET > USINT#0) THEN
                    Pusher$Timer3$ET := (Pusher$Timer3$ET - USINT#1);
                ELSE
                    Pusher$Timer3$ET := USINT#0;
                END_IF
            ELSE
                Pusher$Timer3$Q := FALSE;
                Pusher$Timer3$ET := Pusher$Timer3$PT;
            END_IF
            Pusher$Slide3_white := (Pusher$Slide3_white - INT#1);
            Pusher$Priority_Var_White := (Pusher$Priority_Var_White - INT#1);
            IF TRUE THEN
                Pusher$_transit := TRUE;
                Pusher$_state := Pusher_states_t#Interstep_2;
            END_IF

        Pusher_states_t#Second_Slide_Timer_Black:
            Pusher$_transit := FALSE;
            IF (Pusher$SorterLightnesssensorCraneInterfaceInverse = TRUE) THEN
                Pusher$Timer_Slide2_Black$IN := Pusher$SorterLightnesssensorCraneInterfaceInverse;
                Pusher$Timer_Slide2_Black$PT := Pusher$Duration_Slide2_Black;
                IF Pusher$Timer_Slide2_Black$IN THEN
                    Pusher$Timer_Slide2_Black$Q := (Pusher$Timer_Slide2_Black$ET = USINT#0);
                    IF (Pusher$Timer_Slide2_Black$ET > USINT#0) THEN
                        Pusher$Timer_Slide2_Black$ET := (Pusher$Timer_Slide2_Black$ET - USINT#1);
                    ELSE
                        Pusher$Timer_Slide2_Black$ET := USINT#0;
                    END_IF
                ELSE
                    Pusher$Timer_Slide2_Black$Q := FALSE;
                    Pusher$Timer_Slide2_Black$ET := Pusher$Timer_Slide2_Black$PT;
                END_IF
                Pusher$interconnect_Slide2_Black := Pusher$Timer_Slide2_Black$Q;
            END_IF
            IF Pusher$interconnect_Slide2_Black THEN
                Pusher$_transit := TRUE;
                Pusher$_state := Pusher_states_t#PusherY2_Move_Out_Black;
            END_IF

        Pusher_states_t#Second_Slide_Timer_Metal:
            Pusher$_transit := FALSE;
            Pusher$Timer_Slide2_Metal$IN := TRUE;
            Pusher$Timer_Slide2_Metal$PT := Pusher$Duration_Slide2_Metal;
            IF Pusher$Timer_Slide2_Metal$IN THEN
                Pusher$Timer_Slide2_Metal$Q := (Pusher$Timer_Slide2_Metal$ET = USINT#0);
                IF (Pusher$Timer_Slide2_Metal$ET > USINT#0) THEN
                    Pusher$Timer_Slide2_Metal$ET := (Pusher$Timer_Slide2_Metal$ET - USINT#1);
                ELSE
                    Pusher$Timer_Slide2_Metal$ET := USINT#0;
                END_IF
            ELSE
                Pusher$Timer_Slide2_Metal$Q := FALSE;
                Pusher$Timer_Slide2_Metal$ET := Pusher$Timer_Slide2_Metal$PT;
            END_IF
            Pusher$interconnect_Slide2_Metal := Pusher$Timer_Slide2_Metal$Q;
            IF Pusher$interconnect_Slide2_Metal THEN
                Pusher$_transit := TRUE;
                Pusher$_state := Pusher_states_t#PusherY2_Move_Out_Metal;
            END_IF

        Pusher_states_t#Second_Slide_Timer_White:
            Pusher$_transit := FALSE;
            Pusher$Timer_Slide2_White$IN := TRUE;
            Pusher$Timer_Slide2_White$PT := Pusher$Duration_Slide2_White;
            IF Pusher$Timer_Slide2_White$IN THEN
                Pusher$Timer_Slide2_White$Q := (Pusher$Timer_Slide2_White$ET = USINT#0);
                IF (Pusher$Timer_Slide2_White$ET > USINT#0) THEN
                    Pusher$Timer_Slide2_White$ET := (Pusher$Timer_Slide2_White$ET - USINT#1);
                ELSE
                    Pusher$Timer_Slide2_White$ET := USINT#0;
                END_IF
            ELSE
                Pusher$Timer_Slide2_White$Q := FALSE;
                Pusher$Timer_Slide2_White$ET := Pusher$Timer_Slide2_White$PT;
            END_IF
            Pusher$interconnect_Slide2_White := Pusher$Timer_Slide2_White$Q;
            IF Pusher$interconnect_Slide2_White THEN
                Pusher$_transit := TRUE;
                Pusher$_state := Pusher_states_t#PusherY2_Move_Out_White;
            END_IF

        Pusher_states_t#Second_Slide_black_workpieces:
            Pusher$_transit := FALSE;
            IF TRUE THEN
                Pusher$_transit := TRUE;
                Pusher$_state := Pusher_states_t#Second_Slide_Timer_Black;
            END_IF

        Pusher_states_t#Second_Slide_metal_workpieces:
            Pusher$_transit := FALSE;
            IF (Pusher$SorterLightnessSensorPusher2 AND Pusher$SorterCapacitiveSensorPusher2) THEN
                Pusher$_transit := TRUE;
                Pusher$_state := Pusher_states_t#Second_Test_For_Metal;
            END_IF

        Pusher_states_t#Second_Slide_white_workpieces:
            Pusher$_transit := FALSE;
            IF (Pusher$SorterLightnessSensorPusher2 AND NOT Pusher$SorterCapacitiveSensorPusher2) THEN
                Pusher$_transit := TRUE;
                Pusher$_state := Pusher_states_t#Second_Test_For_White;
            END_IF

        Pusher_states_t#Second_Test_For_Metal:
            Pusher$_transit := FALSE;
            IF TRUE THEN
                Pusher$_transit := TRUE;
                Pusher$_state := Pusher_states_t#Second_Slide_Timer_Metal;
            END_IF

        Pusher_states_t#Second_Test_For_White:
            Pusher$_transit := FALSE;
            IF TRUE THEN
                Pusher$_transit := TRUE;
                Pusher$_state := Pusher_states_t#Second_Slide_Timer_White;
            END_IF

        Pusher_states_t#Third_Slide_black_workpieces:
            Pusher$_transit := FALSE;
            IF (NOT Pusher$SorterLightnessSensorPusher2 AND NOT Pusher$SorterCapacitiveSensorPusher2) THEN
                Pusher$_transit := TRUE;
                Pusher$_state := Pusher_states_t#Wait_Black;
            END_IF

        Pusher_states_t#Third_Slide_metal_workpieces:
            Pusher$_transit := FALSE;
            IF (Pusher$SorterLightnessSensorPusher2 AND Pusher$SorterCapacitiveSensorPusher2) THEN
                Pusher$_transit := TRUE;
                Pusher$_state := Pusher_states_t#Wait_Metal;
            END_IF

        Pusher_states_t#Third_Slide_white_workpieces:
            Pusher$_transit := FALSE;
            IF (Pusher$SorterLightnessSensorPusher2 AND NOT Pusher$SorterCapacitiveSensorPusher2) THEN
                Pusher$_transit := TRUE;
                Pusher$_state := Pusher_states_t#Wait_White;
            END_IF

        Pusher_states_t#Wait_Black:
            Pusher$_transit := FALSE;
            IF ((NOT Pusher$SorterLightnessSensorPusher2 AND NOT Pusher$SorterCapacitiveSensorPusher2) = TRUE) THEN
                Pusher$Timer2$IN := (NOT Pusher$SorterLightnessSensorPusher2 AND NOT Pusher$SorterCapacitiveSensorPusher2);
                Pusher$Timer2$PT := Pusher$Duration2;
                IF Pusher$Timer2$IN THEN
                    Pusher$Timer2$Q := (Pusher$Timer2$ET = USINT#0);
                    IF (Pusher$Timer2$ET > USINT#0) THEN
                        Pusher$Timer2$ET := (Pusher$Timer2$ET - USINT#1);
                    ELSE
                        Pusher$Timer2$ET := USINT#0;
                    END_IF
                ELSE
                    Pusher$Timer2$Q := FALSE;
                    Pusher$Timer2$ET := Pusher$Timer2$PT;
                END_IF
                Pusher$interconnect2 := Pusher$Timer2$Q;
            END_IF
            IF Pusher$interconnect2 THEN
                Pusher$_transit := TRUE;
                Pusher$_state := Pusher_states_t#Reset_interconnect3;
            END_IF

        Pusher_states_t#Wait_Metal:
            Pusher$_transit := FALSE;
            Pusher$Timer3$IN := TRUE;
            Pusher$Timer3$PT := Pusher$Duration3;
            IF Pusher$Timer3$IN THEN
                Pusher$Timer3$Q := (Pusher$Timer3$ET = USINT#0);
                IF (Pusher$Timer3$ET > USINT#0) THEN
                    Pusher$Timer3$ET := (Pusher$Timer3$ET - USINT#1);
                ELSE
                    Pusher$Timer3$ET := USINT#0;
                END_IF
            ELSE
                Pusher$Timer3$Q := FALSE;
                Pusher$Timer3$ET := Pusher$Timer3$PT;
            END_IF
            Pusher$interconnect3 := Pusher$Timer3$Q;
            IF Pusher$interconnect3 THEN
                Pusher$_transit := TRUE;
                Pusher$_state := Pusher_states_t#Reset_interconnect_Slide3_Metal;
            END_IF

        Pusher_states_t#Wait_White:
            Pusher$_transit := FALSE;
            Pusher$Timer3$IN := TRUE;
            Pusher$Timer3$PT := Pusher$Duration3;
            IF Pusher$Timer3$IN THEN
                Pusher$Timer3$Q := (Pusher$Timer3$ET = USINT#0);
                IF (Pusher$Timer3$ET > USINT#0) THEN
                    Pusher$Timer3$ET := (Pusher$Timer3$ET - USINT#1);
                ELSE
                    Pusher$Timer3$ET := USINT#0;
                END_IF
            ELSE
                Pusher$Timer3$Q := FALSE;
                Pusher$Timer3$ET := Pusher$Timer3$PT;
            END_IF
            Pusher$interconnect3 := Pusher$Timer3$Q;
            IF Pusher$interconnect3 THEN
                Pusher$_transit := TRUE;
                Pusher$_state := Pusher_states_t#Reset_interconnect_Slide3_White;
            END_IF
